LIN {X 0,Y 298.848,Z 1149.054,A -85,B 0,C 180,E1 12296.263,E2 12296.263} C_VEL
LIN {X 0,Y 306.631,Z 1138.503,A -85,B 0,C 180,E1 12292.663,E2 12292.663} C_VEL
LIN {X 0,Y 315.41,Z 1126.647,A -85,B 0,C 180,E1 12289.23,E2 12289.23} C_VEL
LIN {X 0,Y 327.193,Z 1110.564,A -85,B 0,C 180,E1 12285.344,E2 12285.344} C_VEL
LIN {X 0,Y 338.522,Z 1094.359,A -85,B 0,C 180,E1 12282.153,E2 12282.153} C_VEL
LIN {X 0,Y 348.344,Z 1079.778,A -85,B 0,C 180,E1 12279.714,E2 12279.714} C_VEL
LIN {X 0,Y 358.568,Z 1063.892,A -85,B 0,C 180,E1 12277.439,E2 12277.439} C_VEL
LIN {X 0,Y 370.942,Z 1043.552,A -85,B 0,C 180,E1 12274.974,E2 12274.974} C_VEL
LIN {X 0,Y 382.686,Z 1022.269,A -85,B 0,C 180,E1 12272.861,E2 12272.861} C_VEL
LIN {X 0,Y 392.079,Z 1003.934,A -85,B 0,C 180,E1 12271.318,E2 12271.318} C_VEL
LIN {X 0,Y 400.638,Z 985.807,A -85,B 0,C 180,E1 12270.004,E2 12270.004} C_VEL
LIN {X 0,Y 409.368,Z 965.527,A -85,B 0,C 180,E1 12268.737,E2 12268.737} C_VEL
LIN {X 0,Y 419.427,Z 939.151,A -85,B 0,C 180,E1 12267.379,E2 12267.379} C_VEL
LIN {X 0,Y 426.63,Z 917.308,A -85,B 0,C 180,E1 12266.458,E2 12266.458} C_VEL
LIN {X 0,Y 432.569,Z 896.655,A -85,B 0,C 180,E1 12265.726,E2 12265.726} C_VEL
LIN {X 0,Y 432.97,Z 895.159,A -85,B 0,C 180,E1 12265.678,E2 12265.678} C_VEL
LIN {X 0,Y 434.572,Z 887.998,A -85,B 0,C 180,E1 12265.339,E2 12265.339} C_VEL
LIN {X 0,Y 436.586,Z 870.292,A -85,B 0,C 180,E1 12264.11,E2 12264.11} C_VEL
LIN {X 0,Y 437.717,Z 862.972,A -85,B 0,C 180,E1 12263.81,E2 12263.81} C_VEL
LIN {X 0,Y 441.966,Z 839.481,A -85,B 0,C 180,E1 12263.335,E2 12263.335} C_VEL
LIN {X 0,Y 444.937,Z 817.163,A -85,B 0,C 180,E1 12262.954,E2 12262.954} C_VEL
LIN {X 0,Y 464.403,Z 606.648,A -85,B 0,C 180,E1 12259.789,E2 12259.789} C_VEL
LIN {X 0,Y 465.771,Z 591.946,A -85,B 0,C 180,E1 12259.566,E2 12259.566} C_VEL
LIN {X 0,Y 461.251,Z 583.723,A -85,B 0,C 180,E1 12256.887,E2 12256.887} C_VEL
LIN {X 0,Y 458.078,Z 578.07,A -85,B 0,C 180,E1 12254.603,E2 12254.603} C_VEL
LIN {X 0,Y 456.376,Z 575.276,A -85,B 0,C 180,E1 12253.171,E2 12253.171} C_VEL
LIN {X 0,Y 454.555,Z 571.903,A -85,B 0,C 180,E1 12251.29,E2 12251.29} C_VEL
LIN {X 0,Y 452.297,Z 567.52,A -85,B 0,C 180,E1 12247.878,E2 12247.878} C_VEL
LIN {X 0,Y 451.171,Z 566.506,A -85,B 0,C 180,E1 12243.176,E2 12243.176} C_VEL
LIN {X 0,Y 452.449,Z 567.778,A -85,B 0,C 180,E1 12238.924,E2 12238.924} C_VEL
LIN {X 0,Y 454.653,Z 571.991,A -85,B 0,C 180,E1 12235.712,E2 12235.712} C_VEL
LIN {X 0,Y 457.727,Z 577.434,A -85,B 0,C 180,E1 12232.784,E2 12232.784} C_VEL
LIN {X 0,Y 461.178,Z 583.607,A -85,B 0,C 180,E1 12230.264,E2 12230.264} C_VEL
LIN {X 0,Y 465.657,Z 591.717,A -85,B 0,C 180,E1 12227.6,E2 12227.6} C_VEL
LIN {X 0,Y 465.809,Z 592.384,A -85,B 0,C 180,E1 12227.497,E2 12227.497} C_VEL
LIN {X 0,Y 445.561,Z 812.948,A -85,B 0,C 180,E1 12224.189,E2 12224.189} C_VEL
LIN {X 0,Y 442.274,Z 839.432,A -85,B 0,C 180,E1 12223.745,E2 12223.745} C_VEL
LIN {X 0,Y 438.393,Z 861.631,A -85,B 0,C 180,E1 12223.316,E2 12223.316} C_VEL
LIN {X 0,Y 433.612,Z 883.484,A -85,B 0,C 180,E1 12222.797,E2 12222.797} C_VEL
LIN {X 0,Y 426.781,Z 909.478,A -85,B 0,C 180,E1 12222.021,E2 12222.021} C_VEL
LIN {X 0,Y 418.611,Z 934.825,A -85,B 0,C 180,E1 12221.058,E2 12221.058} C_VEL
LIN {X 0,Y 411.381,Z 954.622,A -85,B 0,C 180,E1 12220.152,E2 12220.152} C_VEL
LIN {X 0,Y 403.296,Z 974.499,A -85,B 0,C 180,E1 12219.083,E2 12219.083} C_VEL
LIN {X 0,Y 394.183,Z 994.824,A -85,B 0,C 180,E1 12217.793,E2 12217.793} C_VEL
LIN {X 0,Y 382.115,Z 1019.005,A -85,B 0,C 180,E1 12215.952,E2 12215.952} C_VEL
LIN {X 0,Y 371.516,Z 1038.231,A -85,B 0,C 180,E1 12214.189,E2 12214.189} C_VEL
LIN {X 0,Y 361.689,Z 1054.851,A -85,B 0,C 180,E1 12212.41,E2 12212.41} C_VEL
LIN {X 0,Y 351.422,Z 1071.214,A -85,B 0,C 180,E1 12210.366,E2 12210.366} C_VEL
LIN {X 0,Y 339.159,Z 1089.74,A -85,B 0,C 180,E1 12207.631,E2 12207.631} C_VEL
LIN {X 0,Y 326.616,Z 1107.457,A -85,B 0,C 180,E1 12204.432,E2 12204.432} C_VEL
LIN {X 0,Y 316.723,Z 1120.957,A -85,B 0,C 180,E1 12201.527,E2 12201.527} C_VEL
LIN {X 0,Y 307.464,Z 1133.293,A -85,B 0,C 180,E1 12198.413,E2 12198.413} C_VEL
LIN {X 0,Y 298.632,Z 1144.957,A -85,B 0,C 180,E1 12194.947,E2 12194.947} C_VEL
LIN {X 0,Y 288.909,Z 1157.956,A -85,B 0,C 180,E1 12190.328,E2 12190.328} C_VEL
LIN {X 0,Y 280.637,Z 1169.184,A -85,B 0,C 180,E1 12185.322,E2 12185.322} C_VEL
LIN {X 0,Y 275.188,Z 1177.115,A -85,B 0,C 180,E1 12181.06,E2 12181.06} C_VEL
LIN {X 0,Y 270.808,Z 1184.121,A -85,B 0,C 180,E1 12176.535,E2 12176.535} C_VEL
LIN {X 0,Y 267.412,Z 1190.479,A -85,B 0,C 180,E1 12171.495,E2 12171.495} C_VEL
LIN {X 0,Y 265.075,Z 1196.182,A -85,B 0,C 180,E1 12165.534,E2 12165.534} C_VEL
LIN {X 0,Y 264.182,Z 1199.596,A -85,B 0,C 180,E1 12160.467,E2 12160.467} C_VEL
LIN {X 0,Y 263.953,Z 1201.5,A -85,B 0,C 180,E1 12156.307,E2 12156.307} C_VEL
LIN {X 0,Y 263.915,Z 1202.584,A -85,B 0,C 180,E1 12151.954,E2 12151.954} C_VEL
LIN {X 0,Y 263.913,Z 1202.769,A -85,B 0,C 180,E1 12147.829,E2 12147.829} C_VEL
LIN {X 0,Y 263.958,Z 1202.061,A -85,B 0,C 180,E1 12143.475,E2 12143.475} C_VEL
LIN {X 0,Y 264.264,Z 1200.332,A -85,B 0,C 180,E1 12138.874,E2 12138.874} C_VEL
LIN {X 0,Y 265.245,Z 1197.443,A -85,B 0,C 180,E1 12134.027,E2 12134.027} C_VEL
LIN {X 0,Y 267.07,Z 1193.652,A -85,B 0,C 180,E1 12129.388,E2 12129.388} C_VEL
LIN {X 0,Y 269.995,Z 1188.844,A -85,B 0,C 180,E1 12124.794,E2 12124.794} C_VEL
LIN {X 0,Y 274.352,Z 1182.67,A -85,B 0,C 180,E1 12120.047,E2 12120.047} C_VEL
LIN {X 0,Y 281.35,Z 1173.897,A -85,B 0,C 180,E1 12114.601,E2 12114.601} C_VEL
LIN {X 0,Y 290.342,Z 1163.146,A -85,B 0,C 180,E1 12109.393,E2 12109.393} C_VEL
LIN {X 0,Y 299.108,Z 1153.094,A -85,B 0,C 180,E1 12105.401,E2 12105.401} C_VEL
LIN {X 0,Y 308.541,Z 1142.322,A -85,B 0,C 180,E1 12101.812,E2 12101.812} C_VEL
LIN {X 0,Y 320.174,Z 1128.958,A -85,B 0,C 180,E1 12098.098,E2 12098.098} C_VEL
LIN {X 0,Y 334.188,Z 1112.217,A -85,B 0,C 180,E1 12094.334,E2 12094.334} C_VEL
LIN {X 0,Y 346.206,Z 1097.244,A -85,B 0,C 180,E1 12091.573,E2 12091.573} C_VEL
LIN {X 0,Y 357.593,Z 1082.406,A -85,B 0,C 180,E1 12089.264,E2 12089.264} C_VEL
LIN {X 0,Y 369.525,Z 1065.998,A -85,B 0,C 180,E1 12087.101,E2 12087.101} C_VEL
LIN {X 0,Y 384.556,Z 1043.665,A -85,B 0,C 180,E1 12084.673,E2 12084.673} C_VEL
LIN {X 0,Y 395.974,Z 1025.155,A -85,B 0,C 180,E1 12083.018,E2 12083.018} C_VEL
LIN {X 0,Y 405.897,Z 1007.76,A -85,B 0,C 180,E1 12081.686,E2 12081.686} C_VEL
LIN {X 0,Y 415.681,Z 989.14,A -85,B 0,C 180,E1 12080.466,E2 12080.466} C_VEL
LIN {X 0,Y 425.434,Z 968.768,A -85,B 0,C 180,E1 12079.334,E2 12079.334} C_VEL
LIN {X 0,Y 436.603,Z 942.294,A -85,B 0,C 180,E1 12078.125,E2 12078.125} C_VEL
LIN {X 0,Y 444.581,Z 920.371,A -85,B 0,C 180,E1 12077.313,E2 12077.313} C_VEL
LIN {X 0,Y 451.161,Z 899.649,A -85,B 0,C 180,E1 12076.676,E2 12076.676} C_VEL
LIN {X 0,Y 456.952,Z 878.361,A -85,B 0,C 180,E1 12076.135,E2 12076.135} C_VEL
LIN {X 0,Y 462.441,Z 854.005,A -85,B 0,C 180,E1 12075.644,E2 12075.644} C_VEL
LIN {X 0,Y 467.168,Z 825.022,A -85,B 0,C 180,E1 12075.163,E2 12075.163} C_VEL
LIN {X 0,Y 474.721,Z 753.481,A -85,B 0,C 180,E1 12074.115,E2 12074.115} C_VEL
LIN {X 0,Y 489.723,Z 608.892,A -85,B 0,C 180,E1 12072.02,E2 12072.02} C_VEL
LIN {X 0,Y 487.951,Z 605.447,A -85,B 0,C 180,E1 12070.15,E2 12070.15} C_VEL
LIN {X 0,Y 486.244,Z 601.834,A -85,B 0,C 180,E1 12067.562,E2 12067.562} C_VEL
LIN {X 0,Y 485.116,Z 600.297,A -85,B 0,C 180,E1 12063.427,E2 12063.427} C_VEL
LIN {X 0,Y 485.932,Z 601.575,A -85,B 0,C 180,E1 12059.822,E2 12059.822} C_VEL
LIN {X 0,Y 486.458,Z 602.272,A -85,B 0,C 180,E1 12058.822,E2 12058.822} C_VEL
LIN {X 0,Y 488.722,Z 606.921,A -85,B 0,C 180,E1 12055.776,E2 12055.776} C_VEL
LIN {X 0,Y 489.67,Z 609.104,A -85,B 0,C 180,E1 12054.794,E2 12054.794} C_VEL
LIN {X 0,Y 467.761,Z 819.218,A -85,B 0,C 180,E1 12051.761,E2 12051.761} C_VEL
LIN {X 0,Y 464.351,Z 842.109,A -85,B 0,C 180,E1 12051.392,E2 12051.392} C_VEL
LIN {X 0,Y 458.756,Z 869.685,A -85,B 0,C 180,E1 12050.863,E2 12050.863} C_VEL
LIN {X 0,Y 452.233,Z 894.407,A -85,B 0,C 180,E1 12050.238,E2 12050.238} C_VEL
LIN {X 0,Y 445.762,Z 915.186,A -85,B 0,C 180,E1 12049.598,E2 12049.598} C_VEL
LIN {X 0,Y 438.233,Z 936.245,A -85,B 0,C 180,E1 12048.817,E2 12048.817} C_VEL
LIN {X 0,Y 428.413,Z 960.404,A -85,B 0,C 180,E1 12047.738,E2 12047.738} C_VEL
LIN {X 0,Y 417.012,Z 984.563,A -85,B 0,C 180,E1 12046.409,E2 12046.409} C_VEL
LIN {X 0,Y 407.061,Z 1003.571,A -85,B 0,C 180,E1 12045.165,E2 12045.165} C_VEL
LIN {X 0,Y 396.757,Z 1021.657,A -85,B 0,C 180,E1 12043.77,E2 12043.77} C_VEL
LIN {X 0,Y 385.992,Z 1039.101,A -85,B 0,C 180,E1 12042.201,E2 12042.201} C_VEL
LIN {X 0,Y 371.615,Z 1060.6,A -85,B 0,C 180,E1 12039.886,E2 12039.886} C_VEL
LIN {X 0,Y 358.628,Z 1078.377,A -85,B 0,C 180,E1 12037.544,E2 12037.544} C_VEL
LIN {X 0,Y 347.334,Z 1092.999,A -85,B 0,C 180,E1 12035.26,E2 12035.26} C_VEL
LIN {X 0,Y 336.246,Z 1106.691,A -85,B 0,C 180,E1 12032.745,E2 12032.745} C_VEL
LIN {X 0,Y 323.776,Z 1121.525,A -85,B 0,C 180,E1 12029.495,E2 12029.495} C_VEL
LIN {X 0,Y 310.177,Z 1137.009,A -85,B 0,C 180,E1 12025.285,E2 12025.285} C_VEL
LIN {X 0,Y 300.104,Z 1148.266,A -85,B 0,C 180,E1 12021.531,E2 12021.531} C_VEL
LIN {X 0,Y 291.682,Z 1157.706,A -85,B 0,C 180,E1 12017.768,E2 12017.768} C_VEL
LIN {X 0,Y 283.4,Z 1167.233,A -85,B 0,C 180,E1 12013.192,E2 12013.192} C_VEL
LIN {X 0,Y 275.392,Z 1176.9,A -85,B 0,C 180,E1 12007.324,E2 12007.324} C_VEL
LIN {X 0,Y 270.615,Z 1183.268,A -85,B 0,C 180,E1 12002.394,E2 12002.394} C_VEL
LIN {X 0,Y 267.55,Z 1187.968,A -85,B 0,C 180,E1 11997.849,E2 11997.849} C_VEL
LIN {X 0,Y 265.565,Z 1191.67,A -85,B 0,C 180,E1 11993.263,E2 11993.263} C_VEL
LIN {X 0,Y 264.48,Z 1194.36,A -85,B 0,C 180,E1 11988.744,E2 11988.744} C_VEL
LIN {X 0,Y 264.052,Z 1196.046,A -85,B 0,C 180,E1 11984.472,E2 11984.472} C_VEL
LIN {X 0,Y 263.934,Z 1196.873,A -85,B 0,C 180,E1 11980.477,E2 11980.477} C_VEL
LIN {X 0,Y 263.92,Z 1196.969,A -85,B 0,C 180,E1 11976.526,E2 11976.526} C_VEL
LIN {X 0,Y 263.936,Z 1196.281,A -85,B 0,C 180,E1 11972.388,E2 11972.388} C_VEL
LIN {X 0,Y 264.123,Z 1194.682,A -85,B 0,C 180,E1 11968.048,E2 11968.048} C_VEL
LIN {X 0,Y 264.764,Z 1191.92,A -85,B 0,C 180,E1 11963.332,E2 11963.332} C_VEL
LIN {X 0,Y 266.139,Z 1188.198,A -85,B 0,C 180,E1 11958.734,E2 11958.734} C_VEL
LIN {X 0,Y 268.44,Z 1183.501,A -85,B 0,C 180,E1 11954.223,E2 11954.223} C_VEL
LIN {X 0,Y 271.793,Z 1177.722,A -85,B 0,C 180,E1 11949.738,E2 11949.738} C_VEL
LIN {X 0,Y 276.754,Z 1170.251,A -85,B 0,C 180,E1 11944.995,E2 11944.995} C_VEL
LIN {X 0,Y 284.886,Z 1159.006,A -85,B 0,C 180,E1 11939.306,E2 11939.306} C_VEL
LIN {X 0,Y 292.503,Z 1148.942,A -85,B 0,C 180,E1 11935.19,E2 11935.19} C_VEL
LIN {X 0,Y 300.637,Z 1138.364,A -85,B 0,C 180,E1 11931.543,E2 11931.543} C_VEL
LIN {X 0,Y 310.272,Z 1125.864,A -85,B 0,C 180,E1 11927.911,E2 11927.911} C_VEL
LIN {X 0,Y 323.096,Z 1108.838,A -85,B 0,C 180,E1 11923.859,E2 11923.859} C_VEL
LIN {X 0,Y 333.735,Z 1094.099,A -85,B 0,C 180,E1 11920.976,E2 11920.976} C_VEL
LIN {X 0,Y 343.862,Z 1079.484,A -85,B 0,C 180,E1 11918.54,E2 11918.54} C_VEL
LIN {X 0,Y 354.807,Z 1062.9,A -85,B 0,C 180,E1 11916.185,E2 11916.185} C_VEL
LIN {X 0,Y 367.89,Z 1041.698,A -85,B 0,C 180,E1 11913.673,E2 11913.673} C_VEL
LIN {X 0,Y 379.107,Z 1021.786,A -85,B 0,C 180,E1 11911.727,E2 11911.727} C_VEL
LIN {X 0,Y 388.71,Z 1003.39,A -85,B 0,C 180,E1 11910.201,E2 11910.201} C_VEL
LIN {X 0,Y 397.461,Z 985.186,A -85,B 0,C 180,E1 11908.904,E2 11908.904} C_VEL
LIN {X 0,Y 407.502,Z 962.18,A -85,B 0,C 180,E1 11907.503,E2 11907.503} C_VEL
LIN {X 0,Y 417,Z 937.133,A -85,B 0,C 180,E1 11906.266,E2 11906.266} C_VEL
LIN {X 0,Y 423.95,Z 916.256,A -85,B 0,C 180,E1 11905.408,E2 11905.408} C_VEL
LIN {X 0,Y 430,Z 895.421,A -85,B 0,C 180,E1 11904.689,E2 11904.689} C_VEL
LIN {X 0,Y 435.648,Z 872.626,A -85,B 0,C 180,E1 11904.044,E2 11904.044} C_VEL
LIN {X 0,Y 437.717,Z 862.972,A -85,B 0,C 180,E1 11903.81,E2 11903.81} C_VEL
LIN {X 0,Y 438.835,Z 855.588,A -85,B 0,C 180,E1 11903.525,E2 11903.525} C_VEL
LIN {X 0,Y 440.138,Z 836.289,A -85,B 0,C 180,E1 11902.384,E2 11902.384} C_VEL
LIN {X 0,Y 440.881,Z 829.878,A -85,B 0,C 180,E1 11902.177,E2 11902.177} C_VEL
LIN {X 0,Y 444.973,Z 790.912,A -85,B 0,C 180,E1 11901.569,E2 11901.569} C_VEL
LIN {X 0,Y 463.11,Z 597.491,A -85,B 0,C 180,E1 11898.684,E2 11898.684} C_VEL
LIN {X 0,Y 459.071,Z 590.031,A -85,B 0,C 180,E1 11896.123,E2 11896.123} C_VEL
LIN {X 0,Y 456.096,Z 584.401,A -85,B 0,C 180,E1 11893.797,E2 11893.797} C_VEL
LIN {X 0,Y 453.353,Z 579.65,A -85,B 0,C 180,E1 11891.058,E2 11891.058} C_VEL
LIN {X 0,Y 451.257,Z 575.43,A -85,B 0,C 180,E1 11887.768,E2 11887.768} C_VEL
LIN {X 0,Y 450.201,Z 574.441,A -85,B 0,C 180,E1 11883.056,E2 11883.056} C_VEL
LIN {X 0,Y 451.425,Z 575.768,A -85,B 0,C 180,E1 11878.985,E2 11878.985} C_VEL
LIN {X 0,Y 453.984,Z 580.782,A -85,B 0,C 180,E1 11875.326,E2 11875.326} C_VEL
LIN {X 0,Y 456.496,Z 585.256,A -85,B 0,C 180,E1 11872.954,E2 11872.954} C_VEL
LIN {X 0,Y 460.172,Z 591.885,A -85,B 0,C 180,E1 11870.242,E2 11870.242} C_VEL
LIN {X 0,Y 463.183,Z 597.705,A -85,B 0,C 180,E1 11868.373,E2 11868.373} C_VEL
LIN {X 0,Y 442.631,Z 816.279,A -85,B 0,C 180,E1 11865.117,E2 11865.117} C_VEL
LIN {X 0,Y 439.544,Z 840.175,A -85,B 0,C 180,E1 11864.717,E2 11864.717} C_VEL
LIN {X 0,Y 435.587,Z 862.291,A -85,B 0,C 180,E1 11864.295,E2 11864.295} C_VEL
LIN {X 0,Y 430.468,Z 885.146,A -85,B 0,C 180,E1 11863.756,E2 11863.756} C_VEL
LIN {X 0,Y 422.635,Z 913.497,A -85,B 0,C 180,E1 11862.895,E2 11862.895} C_VEL
LIN {X 0,Y 415.288,Z 935.737,A -85,B 0,C 180,E1 11862.05,E2 11862.05} C_VEL
LIN {X 0,Y 407.832,Z 955.7,A -85,B 0,C 180,E1 11861.143,E2 11861.143} C_VEL
LIN {X 0,Y 399.392,Z 975.958,A -85,B 0,C 180,E1 11860.059,E2 11860.059} C_VEL
LIN {X 0,Y 388.385,Z 999.758,A -85,B 0,C 180,E1 11858.535,E2 11858.535} C_VEL
LIN {X 0,Y 376.89,Z 1021.741,A -85,B 0,C 180,E1 11856.814,E2 11856.814} C_VEL
LIN {X 0,Y 367.17,Z 1038.915,A -85,B 0,C 180,E1 11855.235,E2 11855.235} C_VEL
LIN {X 0,Y 357.183,Z 1055.378,A -85,B 0,C 180,E1 11853.475,E2 11853.475} C_VEL
LIN {X 0,Y 346.007,Z 1072.703,A -85,B 0,C 180,E1 11851.302,E2 11851.302} C_VEL
LIN {X 0,Y 331.792,Z 1093.31,A -85,B 0,C 180,E1 11848.171,E2 11848.171} C_VEL
LIN {X 0,Y 320.741,Z 1108.389,A -85,B 0,C 180,E1 11845.384,E2 11845.384} C_VEL
LIN {X 0,Y 310.954,Z 1121.299,A -85,B 0,C 180,E1 11842.573,E2 11842.573} C_VEL
LIN {X 0,Y 301.399,Z 1133.582,A -85,B 0,C 180,E1 11839.436,E2 11839.436} C_VEL
LIN {X 0,Y 291.791,Z 1145.799,A -85,B 0,C 180,E1 11835.738,E2 11835.738} C_VEL
LIN {X 0,Y 280.975,Z 1159.554,A -85,B 0,C 180,E1 11830.633,E2 11830.633} C_VEL
LIN {X 0,Y 273.407,Z 1169.459,A -85,B 0,C 180,E1 11826.07,E2 11826.07} C_VEL
LIN {X 0,Y 267.786,Z 1177.242,A -85,B 0,C 180,E1 11821.767,E2 11821.767} C_VEL
LIN {X 0,Y 263.183,Z 1184.219,A -85,B 0,C 180,E1 11817.122,E2 11817.122} C_VEL
LIN {X 0,Y 259.356,Z 1191.071,A -85,B 0,C 180,E1 11811.484,E2 11811.484} C_VEL
LIN {X 0,Y 257.071,Z 1196.358,A -85,B 0,C 180,E1 11805.567,E2 11805.567} C_VEL
LIN {X 0,Y 256.213,Z 1199.464,A -85,B 0,C 180,E1 11800.796,E2 11800.796} C_VEL
LIN {X 0,Y 255.953,Z 1201.455,A -85,B 0,C 180,E1 11796.279,E2 11796.279} C_VEL
LIN {X 0,Y 255.915,Z 1202.488,A -85,B 0,C 180,E1 11792.015,E2 11792.015} C_VEL
LIN {X 0,Y 255.913,Z 1202.689,A -85,B 0,C 180,E1 11787.761,E2 11787.761} C_VEL
LIN {X 0,Y 255.97,Z 1201.929,A -85,B 0,C 180,E1 11783.045,E2 11783.045} C_VEL
LIN {X 0,Y 256.334,Z 1200.153,A -85,B 0,C 180,E1 11778.262,E2 11778.262} C_VEL
LIN {X 0,Y 257.38,Z 1197.414,A -85,B 0,C 180,E1 11773.526,E2 11773.526} C_VEL
LIN {X 0,Y 259.356,Z 1193.649,A -85,B 0,C 180,E1 11768.753,E2 11768.753} C_VEL
LIN {X 0,Y 262.509,Z 1188.849,A -85,B 0,C 180,E1 11764.017,E2 11764.017} C_VEL
LIN {X 0,Y 266.91,Z 1183.002,A -85,B 0,C 180,E1 11759.372,E2 11759.372} C_VEL
LIN {X 0,Y 272.969,Z 1175.708,A -85,B 0,C 180,E1 11754.638,E2 11754.638} C_VEL
LIN {X 0,Y 282.438,Z 1165.063,A -85,B 0,C 180,E1 11749.087,E2 11749.087} C_VEL
LIN {X 0,Y 292.714,Z 1153.752,A -85,B 0,C 180,E1 11744.447,E2 11744.447} C_VEL
LIN {X 0,Y 302.503,Z 1143.04,A -85,B 0,C 180,E1 11740.808,E2 11740.808} C_VEL
LIN {X 0,Y 313.371,Z 1131.023,A -85,B 0,C 180,E1 11737.395,E2 11737.395} C_VEL
LIN {X 0,Y 327.077,Z 1115.493,A -85,B 0,C 180,E1 11733.748,E2 11733.748} C_VEL
LIN {X 0,Y 341.275,Z 1098.356,A -85,B 0,C 180,E1 11730.532,E2 11730.532} C_VEL
LIN {X 0,Y 352.932,Z 1083.631,A -85,B 0,C 180,E1 11728.229,E2 11728.229} C_VEL
LIN {X 0,Y 364.759,Z 1067.847,A -85,B 0,C 180,E1 11726.14,E2 11726.14} C_VEL
LIN {X 0,Y 377.427,Z 1049.832,A -85,B 0,C 180,E1 11724.129,E2 11724.129} C_VEL
LIN {X 0,Y 391.698,Z 1027.619,A -85,B 0,C 180,E1 11722.089,E2 11722.089} C_VEL
LIN {X 0,Y 402.823,Z 1008.606,A -85,B 0,C 180,E1 11720.639,E2 11720.639} C_VEL
LIN {X 0,Y 412.937,Z 989.771,A -85,B 0,C 180,E1 11719.42,E2 11719.42} C_VEL
LIN {X 0,Y 422.517,Z 970.179,A -85,B 0,C 180,E1 11718.346,E2 11718.346} C_VEL
LIN {X 0,Y 433.351,Z 945.415,A -85,B 0,C 180,E1 11717.214,E2 11717.214} C_VEL
LIN {X 0,Y 442.286,Z 921.417,A -85,B 0,C 180,E1 11716.332,E2 11716.332} C_VEL
LIN {X 0,Y 449.171,Z 900.148,A -85,B 0,C 180,E1 11715.689,E2 11715.689} C_VEL
LIN {X 0,Y 455.048,Z 878.936,A -85,B 0,C 180,E1 11715.16,E2 11715.16} C_VEL
LIN {X 0,Y 460.325,Z 856.02,A -85,B 0,C 180,E1 11714.705,E2 11714.705} C_VEL
LIN {X 0,Y 465.493,Z 825.554,A -85,B 0,C 180,E1 11714.204,E2 11714.204} C_VEL
LIN {X 0,Y 472.341,Z 762.313,A -85,B 0,C 180,E1 11713.286,E2 11713.286} C_VEL
LIN {X 0,Y 487.877,Z 615.419,A -85,B 0,C 180,E1 11711.197,E2 11711.197} C_VEL
LIN {X 0,Y 486.678,Z 613.023,A -85,B 0,C 180,E1 11709.818,E2 11709.818} C_VEL
LIN {X 0,Y 485.205,Z 609.734,A -85,B 0,C 180,E1 11707.46,E2 11707.46} C_VEL
LIN {X 0,Y 484.142,Z 608.225,A -85,B 0,C 180,E1 11703.315,E2 11703.315} C_VEL
LIN {X 0,Y 485.295,Z 609.813,A -85,B 0,C 180,E1 11699.174,E2 11699.174} C_VEL
LIN {X 0,Y 487.562,Z 614.715,A -85,B 0,C 180,E1 11695.943,E2 11695.943} C_VEL
LIN {X 0,Y 487.815,Z 615.548,A -85,B 0,C 180,E1 11695.636,E2 11695.636} C_VEL
LIN {X 0,Y 465.995,Z 820.655,A -85,B 0,C 180,E1 11692.706,E2 11692.706} C_VEL
LIN {X 0,Y 462.095,Z 845.781,A -85,B 0,C 180,E1 11692.304,E2 11692.304} C_VEL
LIN {X 0,Y 455.964,Z 873.94,A -85,B 0,C 180,E1 11691.751,E2 11691.751} C_VEL
LIN {X 0,Y 449.996,Z 895.916,A -85,B 0,C 180,E1 11691.197,E2 11691.197} C_VEL
LIN {X 0,Y 443.429,Z 916.521,A -85,B 0,C 180,E1 11690.57,E2 11690.57} C_VEL
LIN {X 0,Y 435.816,Z 937.363,A -85,B 0,C 180,E1 11689.807,E2 11689.807} C_VEL
LIN {X 0,Y 425.211,Z 962.757,A -85,B 0,C 180,E1 11688.68,E2 11688.68} C_VEL
LIN {X 0,Y 414.342,Z 985.231,A -85,B 0,C 180,E1 11687.456,E2 11687.456} C_VEL
LIN {X 0,Y 404.08,Z 1004.424,A -85,B 0,C 180,E1 11686.216,E2 11686.216} C_VEL
LIN {X 0,Y 393.469,Z 1022.632,A -85,B 0,C 180,E1 11684.826,E2 11684.826} C_VEL
LIN {X 0,Y 380.591,Z 1042.975,A -85,B 0,C 180,E1 11682.993,E2 11682.993} C_VEL
LIN {X 0,Y 366.412,Z 1063.233,A -85,B 0,C 180,E1 11680.762,E2 11680.762} C_VEL
LIN {X 0,Y 354.454,Z 1079.15,A -85,B 0,C 180,E1 11678.66,E2 11678.66} C_VEL
LIN {X 0,Y 342.721,Z 1093.899,A -85,B 0,C 180,E1 11676.357,E2 11676.357} C_VEL
LIN {X 0,Y 330.129,Z 1108.948,A -85,B 0,C 180,E1 11673.562,E2 11673.562} C_VEL
LIN {X 0,Y 315.133,Z 1125.965,A -85,B 0,C 180,E1 11669.655,E2 11669.655} C_VEL
LIN {X 0,Y 304.036,Z 1138.054,A -85,B 0,C 180,E1 11666.234,E2 11666.234} C_VEL
LIN {X 0,Y 294.231,Z 1148.574,A -85,B 0,C 180,E1 11662.672,E2 11662.672} C_VEL
LIN {X 0,Y 284.993,Z 1158.455,A -85,B 0,C 180,E1 11658.659,E2 11658.659} C_VEL
LIN {X 0,Y 275.319,Z 1169.106,A -85,B 0,C 180,E1 11653.344,E2 11653.344} C_VEL
LIN {X 0,Y 267.721,Z 1177.73,A -85,B 0,C 180,E1 11647.77,E2 11647.77} C_VEL
LIN {X 0,Y 262.966,Z 1183.719,A -85,B 0,C 180,E1 11642.937,E2 11642.937} C_VEL
LIN {X 0,Y 259.61,Z 1188.559,A -85,B 0,C 180,E1 11638.026,E2 11638.026} C_VEL
LIN {X 0,Y 257.357,Z 1192.611,A -85,B 0,C 180,E1 11632.62,E2 11632.62} C_VEL
LIN {X 0,Y 256.215,Z 1195.623,A -85,B 0,C 180,E1 11626.551,E2 11626.551} C_VEL
LIN {X 0,Y 255.946,Z 1196.882,A -85,B 0,C 180,E1 11621.492,E2 11621.492} C_VEL
LIN {X 0,Y 255.925,Z 1197.094,A -85,B 0,C 180,E1 11616.956,E2 11616.956} C_VEL
LIN {X 0,Y 255.936,Z 1196.409,A -85,B 0,C 180,E1 11612.463,E2 11612.463} C_VEL
LIN {X 0,Y 256.147,Z 1194.724,A -85,B 0,C 180,E1 11607.763,E2 11607.763} C_VEL
LIN {X 0,Y 256.815,Z 1192.063,A -85,B 0,C 180,E1 11603.068,E2 11603.068} C_VEL
LIN {X 0,Y 258.255,Z 1188.409,A -85,B 0,C 180,E1 11598.386,E2 11598.386} C_VEL
LIN {X 0,Y 260.689,Z 1183.74,A -85,B 0,C 180,E1 11593.741,E2 11593.741} C_VEL
LIN {X 0,Y 264.193,Z 1178.029,A -85,B 0,C 180,E1 11589.161,E2 11589.161} C_VEL
LIN {X 0,Y 269.169,Z 1170.891,A -85,B 0,C 180,E1 11584.476,E2 11584.476} C_VEL
LIN {X 0,Y 277.115,Z 1160.456,A -85,B 0,C 180,E1 11578.939,E2 11578.939} C_VEL
LIN {X 0,Y 285.952,Z 1149.215,A -85,B 0,C 180,E1 11574.217,E2 11574.217} C_VEL
LIN {X 0,Y 294.316,Z 1138.783,A -85,B 0,C 180,E1 11570.559,E2 11570.559} C_VEL
LIN {X 0,Y 303.298,Z 1127.554,A -85,B 0,C 180,E1 11567.227,E2 11567.227} C_VEL
LIN {X 0,Y 314.946,Z 1112.769,A -85,B 0,C 180,E1 11563.546,E2 11563.546} C_VEL
LIN {X 0,Y 328.02,Z 1095.319,A -85,B 0,C 180,E1 11560.03,E2 11560.03} C_VEL
LIN {X 0,Y 338.898,Z 1080.087,A -85,B 0,C 180,E1 11557.474,E2 11557.474} C_VEL
LIN {X 0,Y 349.516,Z 1064.448,A -85,B 0,C 180,E1 11555.242,E2 11555.242} C_VEL
LIN {X 0,Y 361.981,Z 1044.961,A -85,B 0,C 180,E1 11552.892,E2 11552.892} C_VEL
LIN {X 0,Y 374.609,Z 1023.252,A -85,B 0,C 180,E1 11550.746,E2 11550.746} C_VEL
LIN {X 0,Y 384.761,Z 1004.269,A -85,B 0,C 180,E1 11549.174,E2 11549.174} C_VEL
LIN {X 0,Y 393.679,Z 986.144,A -85,B 0,C 180,E1 11547.891,E2 11547.891} C_VEL
LIN {X 0,Y 402.747,Z 965.871,A -85,B 0,C 180,E1 11546.654,E2 11546.654} C_VEL
LIN {X 0,Y 413.177,Z 939.527,A -85,B 0,C 180,E1 11545.333,E2 11545.333} C_VEL
LIN {X 0,Y 420.722,Z 917.399,A -85,B 0,C 180,E1 11544.427,E2 11544.427} C_VEL
LIN {X 0,Y 426.971,Z 896.339,A -85,B 0,C 180,E1 11543.706,E2 11543.706} C_VEL
LIN {X 0,Y 432.496,Z 874.558,A -85,B 0,C 180,E1 11543.093,E2 11543.093} C_VEL
LIN {X 0,Y 438.082,Z 847.644,A -85,B 0,C 180,E1 11542.494,E2 11542.494} C_VEL
LIN {X 0,Y 440.881,Z 829.878,A -85,B 0,C 180,E1 11542.177,E2 11542.177} C_VEL
LIN {X 0,Y 441.632,Z 822.395,A -85,B 0,C 180,E1 11541.928,E2 11541.928} C_VEL
LIN {X 0,Y 441.723,Z 802.826,A -85,B 0,C 180,E1 11540.851,E2 11540.851} C_VEL
LIN {X 0,Y 442.089,Z 796.338,A -85,B 0,C 180,E1 11540.659,E2 11540.659} C_VEL
LIN {X 0,Y 460.588,Z 603.061,A -85,B 0,C 180,E1 11537.808,E2 11537.808} C_VEL
LIN {X 0,Y 456.266,Z 594.858,A -85,B 0,C 180,E1 11534.792,E2 11534.792} C_VEL
LIN {X 0,Y 454.147,Z 591.116,A -85,B 0,C 180,E1 11532.978,E2 11532.978} C_VEL
LIN {X 0,Y 452.165,Z 587.403,A -85,B 0,C 180,E1 11530.834,E2 11530.834} C_VEL
LIN {X 0,Y 450.219,Z 583.341,A -85,B 0,C 180,E1 11527.658,E2 11527.658} C_VEL
LIN {X 0,Y 449.223,Z 582.381,A -85,B 0,C 180,E1 11523.062,E2 11523.062} C_VEL
LIN {X 0,Y 450.375,Z 583.654,A -85,B 0,C 180,E1 11519.11,E2 11519.11} C_VEL
LIN {X 0,Y 452.817,Z 588.579,A -85,B 0,C 180,E1 11515.504,E2 11515.504} C_VEL
LIN {X 0,Y 455.269,Z 593.076,A -85,B 0,C 180,E1 11513.125,E2 11513.125} C_VEL
LIN {X 0,Y 458.785,Z 599.602,A -85,B 0,C 180,E1 11510.466,E2 11510.466} C_VEL
LIN {X 0,Y 460.626,Z 603.453,A -85,B 0,C 180,E1 11509.253,E2 11509.253} C_VEL
LIN {X 0,Y 439.895,Z 818.941,A -85,B 0,C 180,E1 11506.068,E2 11506.068} C_VEL
LIN {X 0,Y 436.866,Z 841.391,A -85,B 0,C 180,E1 11505.693,E2 11505.693} C_VEL
LIN {X 0,Y 432.699,Z 863.996,A -85,B 0,C 180,E1 11505.264,E2 11505.264} C_VEL
LIN {X 0,Y 426.438,Z 890.854,A -85,B 0,C 180,E1 11504.623,E2 11504.623} C_VEL
LIN {X 0,Y 419.065,Z 916.036,A -85,B 0,C 180,E1 11503.838,E2 11503.838} C_VEL
LIN {X 0,Y 412.287,Z 936.096,A -85,B 0,C 180,E1 11503.08,E2 11503.08} C_VEL
LIN {X 0,Y 404.714,Z 955.994,A -85,B 0,C 180,E1 11502.189,E2 11502.189} C_VEL
LIN {X 0,Y 395.826,Z 976.906,A -85,B 0,C 180,E1 11501.082,E2 11501.082} C_VEL
LIN {X 0,Y 383.888,Z 1001.901,A -85,B 0,C 180,E1 11499.479,E2 11499.479} C_VEL
LIN {X 0,Y 373.292,Z 1021.739,A -85,B 0,C 180,E1 11497.934,E2 11497.934} C_VEL
LIN {X 0,Y 363.397,Z 1038.84,A -85,B 0,C 180,E1 11496.379,E2 11496.379} C_VEL
LIN {X 0,Y 352.805,Z 1055.899,A -85,B 0,C 180,E1 11494.568,E2 11494.568} C_VEL
LIN {X 0,Y 340.964,Z 1073.776,A -85,B 0,C 180,E1 11492.325,E2 11492.325} C_VEL
LIN {X 0,Y 326.685,Z 1093.812,A -85,B 0,C 180,E1 11489.26,E2 11489.26} C_VEL
LIN {X 0,Y 315.396,Z 1108.751,A -85,B 0,C 180,E1 11486.486,E2 11486.486} C_VEL
LIN {X 0,Y 305.198,Z 1121.76,A -85,B 0,C 180,E1 11483.63,E2 11483.63} C_VEL
LIN {X 0,Y 294.912,Z 1134.518,A -85,B 0,C 180,E1 11480.319,E2 11480.319} C_VEL
LIN {X 0,Y 283.177,Z 1148.921,A -85,B 0,C 180,E1 11475.788,E2 11475.788} C_VEL
LIN {X 0,Y 273.312,Z 1160.836,A -85,B 0,C 180,E1 11471.093,E2 11471.093} C_VEL
LIN {X 0,Y 266.253,Z 1169.693,A -85,B 0,C 180,E1 11466.879,E2 11466.879} C_VEL
LIN {X 0,Y 260.133,Z 1177.778,A -85,B 0,C 180,E1 11462.26,E2 11462.26} C_VEL
LIN {X 0,Y 254.647,Z 1185.868,A -85,B 0,C 180,E1 11456.591,E2 11456.591} C_VEL
LIN {X 0,Y 250.81,Z 1192.492,A -85,B 0,C 180,E1 11450.469,E2 11450.469} C_VEL
LIN {X 0,Y 249.042,Z 1196.599,A -85,B 0,C 180,E1 11445.508,E2 11445.508} C_VEL
LIN {X 0,Y 248.199,Z 1199.564,A -85,B 0,C 180,E1 11440.679,E2 11440.679} C_VEL
LIN {X 0,Y 247.952,Z 1201.411,A -85,B 0,C 180,E1 11436.25,E2 11436.25} C_VEL
LIN {X 0,Y 247.916,Z 1202.415,A -85,B 0,C 180,E1 11431.849,E2 11431.849} C_VEL
LIN {X 0,Y 247.914,Z 1202.587,A -85,B 0,C 180,E1 11427.457,E2 11427.457} C_VEL
LIN {X 0,Y 247.982,Z 1201.832,A -85,B 0,C 180,E1 11422.703,E2 11422.703} C_VEL
LIN {X 0,Y 248.378,Z 1200.125,A -85,B 0,C 180,E1 11417.917,E2 11417.917} C_VEL
LIN {X 0,Y 249.532,Z 1197.387,A -85,B 0,C 180,E1 11412.992,E2 11412.992} C_VEL
LIN {X 0,Y 251.681,Z 1193.64,A -85,B 0,C 180,E1 11408.072,E2 11408.072} C_VEL
LIN {X 0,Y 255.063,Z 1188.866,A -85,B 0,C 180,E1 11403.205,E2 11403.205} C_VEL
LIN {X 0,Y 259.765,Z 1183.036,A -85,B 0,C 180,E1 11398.434,E2 11398.434} C_VEL
LIN {X 0,Y 266.457,Z 1175.478,A -85,B 0,C 180,E1 11393.422,E2 11393.422} C_VEL
LIN {X 0,Y 276.996,Z 1164.257,A -85,B 0,C 180,E1 11387.546,E2 11387.546} C_VEL
LIN {X 0,Y 286.9,Z 1153.879,A -85,B 0,C 180,E1 11383.25,E2 11383.25} C_VEL
LIN {X 0,Y 297.092,Z 1143.197,A -85,B 0,C 180,E1 11379.584,E2 11379.584} C_VEL
LIN {X 0,Y 308.323,Z 1131.252,A -85,B 0,C 180,E1 11376.173,E2 11376.173} C_VEL
LIN {X 0,Y 322.528,Z 1115.722,A -85,B 0,C 180,E1 11372.519,E2 11372.519} C_VEL
LIN {X 0,Y 337.361,Z 1098.377,A -85,B 0,C 180,E1 11369.277,E2 11369.277} C_VEL
LIN {X 0,Y 349.106,Z 1083.948,A -85,B 0,C 180,E1 11367.037,E2 11367.037} C_VEL
LIN {X 0,Y 361.216,Z 1068.207,A -85,B 0,C 180,E1 11364.97,E2 11364.97} C_VEL
LIN {X 0,Y 373.387,Z 1051.325,A -85,B 0,C 180,E1 11363.1,E2 11363.1} C_VEL
LIN {X 0,Y 388.321,Z 1028.779,A -85,B 0,C 180,E1 11361.034,E2 11361.034} C_VEL
LIN {X 0,Y 400.029,Z 1009.208,A -85,B 0,C 180,E1 11359.559,E2 11359.559} C_VEL
LIN {X 0,Y 410.333,Z 990.402,A -85,B 0,C 180,E1 11358.361,E2 11358.361} C_VEL
LIN {X 0,Y 419.979,Z 971.067,A -85,B 0,C 180,E1 11357.317,E2 11357.317} C_VEL
LIN {X 0,Y 429.762,Z 949.256,A -85,B 0,C 180,E1 11356.327,E2 11356.327} C_VEL
LIN {X 0,Y 440.121,Z 922.475,A -85,B 0,C 180,E1 11355.341,E2 11355.341} C_VEL
LIN {X 0,Y 447.315,Z 900.653,A -85,B 0,C 180,E1 11354.693,E2 11354.693} C_VEL
LIN {X 0,Y 453.277,Z 879.51,A -85,B 0,C 180,E1 11354.178,E2 11354.178} C_VEL
LIN {X 0,Y 458.479,Z 857.369,A -85,B 0,C 180,E1 11353.745,E2 11353.745} C_VEL
LIN {X 0,Y 463.544,Z 829.309,A -85,B 0,C 180,E1 11353.286,E2 11353.286} C_VEL
LIN {X 0,Y 468.817,Z 782.998,A -85,B 0,C 180,E1 11352.617,E2 11352.617} C_VEL
LIN {X 0,Y 486.123,Z 621.802,A -85,B 0,C 180,E1 11350.342,E2 11350.342} C_VEL
LIN {X 0,Y 484.168,Z 617.634,A -85,B 0,C 180,E1 11347.356,E2 11347.356} C_VEL
LIN {X 0,Y 483.164,Z 616.167,A -85,B 0,C 180,E1 11343.322,E2 11343.322} C_VEL
LIN {X 0,Y 484.304,Z 617.846,A -85,B 0,C 180,E1 11339.172,E2 11339.172} C_VEL
LIN {X 0,Y 486.085,Z 621.826,A -85,B 0,C 180,E1 11336.486,E2 11336.486} C_VEL
LIN {X 0,Y 464.517,Z 820.856,A -85,B 0,C 180,E1 11333.676,E2 11333.676} C_VEL
LIN {X 0,Y 460.484,Z 846.396,A -85,B 0,C 180,E1 11333.275,E2 11333.275} C_VEL
LIN {X 0,Y 454.326,Z 874.176,A -85,B 0,C 180,E1 11332.741,E2 11332.741} C_VEL
LIN {X 0,Y 448.56,Z 895.204,A -85,B 0,C 180,E1 11332.224,E2 11332.224} C_VEL
LIN {X 0,Y 441.911,Z 915.887,A -85,B 0,C 180,E1 11331.615,E2 11331.615} C_VEL
LIN {X 0,Y 434.412,Z 936.226,A -85,B 0,C 180,E1 11330.895,E2 11330.895} C_VEL
LIN {X 0,Y 425.022,Z 958.68,A -85,B 0,C 180,E1 11329.941,E2 11329.941} C_VEL
LIN {X 0,Y 413.018,Z 983.603,A -85,B 0,C 180,E1 11328.651,E2 11328.651} C_VEL
LIN {X 0,Y 402.168,Z 1003.655,A -85,B 0,C 180,E1 11327.393,E2 11327.393} C_VEL
LIN {X 0,Y 392.086,Z 1020.733,A -85,B 0,C 180,E1 11326.13,E2 11326.13} C_VEL
LIN {X 0,Y 380.842,Z 1038.283,A -85,B 0,C 180,E1 11324.623,E2 11324.623} C_VEL
LIN {X 0,Y 366.44,Z 1059.088,A -85,B 0,C 180,E1 11322.484,E2 11322.484} C_VEL
LIN {X 0,Y 351.876,Z 1078.1,A -85,B 0,C 180,E1 11320.063,E2 11320.063} C_VEL
LIN {X 0,Y 339.326,Z 1093.496,A -85,B 0,C 180,E1 11317.703,E2 11317.703} C_VEL
LIN {X 0,Y 326.688,Z 1108.18,A -85,B 0,C 180,E1 11315.015,E2 11315.015} C_VEL
LIN {X 0,Y 312.056,Z 1124.375,A -85,B 0,C 180,E1 11311.392,E2 11311.392} C_VEL
LIN {X 0,Y 299.365,Z 1137.679,A -85,B 0,C 180,E1 11307.672,E2 11307.672} C_VEL
LIN {X 0,Y 288.991,Z 1148.354,A -85,B 0,C 180,E1 11304.057,E2 11304.057} C_VEL
LIN {X 0,Y 279.734,Z 1157.801,A -85,B 0,C 180,E1 11300.217,E2 11300.217} C_VEL
LIN {X 0,Y 270.882,Z 1166.921,A -85,B 0,C 180,E1 11295.731,E2 11295.731} C_VEL
LIN {X 0,Y 261.465,Z 1177.021,A -85,B 0,C 180,E1 11289.405,E2 11289.405} C_VEL
LIN {X 0,Y 255.969,Z 1183.397,A -85,B 0,C 180,E1 11284.228,E2 11284.228} C_VEL
LIN {X 0,Y 252.301,Z 1188.196,A -85,B 0,C 180,E1 11279.322,E2 11279.322} C_VEL
LIN {X 0,Y 249.914,Z 1191.963,A -85,B 0,C 180,E1 11274.336,E2 11274.336} C_VEL
LIN {X 0,Y 248.605,Z 1194.63,A -85,B 0,C 180,E1 11269.5,E2 11269.5} C_VEL
LIN {X 0,Y 248.088,Z 1196.278,A -85,B 0,C 180,E1 11264.948,E2 11264.948} C_VEL
LIN {X 0,Y 247.936,Z 1197.067,A -85,B 0,C 180,E1 11260.691,E2 11260.691} C_VEL
LIN {X 0,Y 247.921,Z 1197.126,A -85,B 0,C 180,E1 11256.484,E2 11256.484} C_VEL
LIN {X 0,Y 247.942,Z 1196.401,A -85,B 0,C 180,E1 11252.08,E2 11252.08} C_VEL
LIN {X 0,Y 248.173,Z 1194.767,A -85,B 0,C 180,E1 11247.46,E2 11247.46} C_VEL
LIN {X 0,Y 248.91,Z 1192.087,A -85,B 0,C 180,E1 11242.615,E2 11242.615} C_VEL
LIN {X 0,Y 250.478,Z 1188.415,A -85,B 0,C 180,E1 11237.786,E2 11237.786} C_VEL
LIN {X 0,Y 253.176,Z 1183.608,A -85,B 0,C 180,E1 11232.893,E2 11232.893} C_VEL
LIN {X 0,Y 257.071,Z 1177.703,A -85,B 0,C 180,E1 11228.076,E2 11228.076} C_VEL
LIN {X 0,Y 263.028,Z 1169.745,A -85,B 0,C 180,E1 11222.817,E2 11222.817} C_VEL
LIN {X 0,Y 271.607,Z 1159.018,A -85,B 0,C 180,E1 11217.238,E2 11217.238} C_VEL
LIN {X 0,Y 280.13,Z 1148.71,A -85,B 0,C 180,E1 11212.9,E2 11212.9} C_VEL
LIN {X 0,Y 289.025,Z 1138.081,A -85,B 0,C 180,E1 11209.169,E2 11209.169} C_VEL
LIN {X 0,Y 300.002,Z 1124.904,A -85,B 0,C 180,E1 11205.314,E2 11205.314} C_VEL
LIN {X 0,Y 313.243,Z 1108.381,A -85,B 0,C 180,E1 11201.4,E2 11201.4} C_VEL
LIN {X 0,Y 323.986,Z 1094.396,A -85,B 0,C 180,E1 11198.668,E2 11198.668} C_VEL
LIN {X 0,Y 334.704,Z 1079.783,A -85,B 0,C 180,E1 11196.238,E2 11196.238} C_VEL
LIN {X 0,Y 345.953,Z 1063.611,A -85,B 0,C 180,E1 11193.956,E2 11193.956} C_VEL
LIN {X 0,Y 359.194,Z 1043.303,A -85,B 0,C 180,E1 11191.557,E2 11191.557} C_VEL
LIN {X 0,Y 371.682,Z 1022.104,A -85,B 0,C 180,E1 11189.513,E2 11189.513} C_VEL
LIN {X 0,Y 381.683,Z 1003.713,A -85,B 0,C 180,E1 11188.018,E2 11188.018} C_VEL
LIN {X 0,Y 391.17,Z 984.724,A -85,B 0,C 180,E1 11186.704,E2 11186.704} C_VEL
LIN {X 0,Y 401.989,Z 960.706,A -85,B 0,C 180,E1 11185.295,E2 11185.295} C_VEL
LIN {X 0,Y 411.44,Z 936.386,A -85,B 0,C 180,E1 11184.145,E2 11184.145} C_VEL
LIN {X 0,Y 418.446,Z 915.936,A -85,B 0,C 180,E1 11183.335,E2 11183.335} C_VEL
LIN {X 0,Y 424.68,Z 895.083,A -85,B 0,C 180,E1 11182.644,E2 11182.644} C_VEL
LIN {X 0,Y 430.892,Z 870.599,A -85,B 0,C 180,E1 11181.982,E2 11181.982} C_VEL
LIN {X 0,Y 436.437,Z 842.374,A -85,B 0,C 180,E1 11181.4,E2 11181.4} C_VEL
LIN {X 0,Y 439.709,Z 819.333,A -85,B 0,C 180,E1 11181.012,E2 11181.012} C_VEL
LIN {X 0,Y 442.089,Z 796.338,A -85,B 0,C 180,E1 11180.659,E2 11180.659} C_VEL
LIN {X 0,Y 442.508,Z 788.801,A -85,B 0,C 180,E1 11180.422,E2 11180.422} C_VEL
LIN {X 0,Y 442.645,Z 769.219,A -85,B 0,C 180,E1 11179.355,E2 11179.355} C_VEL
LIN {X 0,Y 443.071,Z 762.736,A -85,B 0,C 180,E1 11179.166,E2 11179.166} C_VEL
LIN {X 0,Y 458.13,Z 608.831,A -85,B 0,C 180,E1 11176.915,E2 11176.915} C_VEL
LIN {X 0,Y 454.431,Z 601.61,A -85,B 0,C 180,E1 11174.137,E2 11174.137} C_VEL
LIN {X 0,Y 452.706,Z 598.502,A -85,B 0,C 180,E1 11172.566,E2 11172.566} C_VEL
LIN {X 0,Y 450.982,Z 595.151,A -85,B 0,C 180,E1 11170.604,E2 11170.604} C_VEL
LIN {X 0,Y 449.182,Z 591.251,A -85,B 0,C 180,E1 11167.547,E2 11167.547} C_VEL
LIN {X 0,Y 448.246,Z 590.321,A -85,B 0,C 180,E1 11163.069,E2 11163.069} C_VEL
LIN {X 0,Y 449.327,Z 591.539,A -85,B 0,C 180,E1 11159.235,E2 11159.235} C_VEL
LIN {X 0,Y 451.655,Z 596.375,A -85,B 0,C 180,E1 11155.683,E2 11155.683} C_VEL
LIN {X 0,Y 453.995,Z 600.789,A -85,B 0,C 180,E1 11153.343,E2 11153.343} C_VEL
LIN {X 0,Y 457.405,Z 607.316,A -85,B 0,C 180,E1 11150.691,E2 11150.691} C_VEL
LIN {X 0,Y 458.172,Z 609.169,A -85,B 0,C 180,E1 11150.144,E2 11150.144} C_VEL
LIN {X 0,Y 437.46,Z 820.026,A -85,B 0,C 180,E1 11147.055,E2 11147.055} C_VEL
LIN {X 0,Y 434.359,Z 842.299,A -85,B 0,C 180,E1 11146.686,E2 11146.686} C_VEL
LIN {X 0,Y 429.842,Z 866.133,A -85,B 0,C 180,E1 11146.237,E2 11146.237} C_VEL
LIN {X 0,Y 422.827,Z 894.666,A -85,B 0,C 180,E1 11145.544,E2 11145.544} C_VEL
LIN {X 0,Y 416.128,Z 916.987,A -85,B 0,C 180,E1 11144.85,E2 11144.85} C_VEL
LIN {X 0,Y 409.112,Z 937.298,A -85,B 0,C 180,E1 11144.091,E2 11144.091} C_VEL
LIN {X 0,Y 401.108,Z 957.824,A -85,B 0,C 180,E1 11143.178,E2 11143.178} C_VEL
LIN {X 0,Y 390.337,Z 982.394,A -85,B 0,C 180,E1 11141.864,E2 11141.864} C_VEL
LIN {X 0,Y 378.964,Z 1005.032,A -85,B 0,C 180,E1 11140.374,E2 11140.374} C_VEL
LIN {X 0,Y 368.947,Z 1023.29,A -85,B 0,C 180,E1 11138.944,E2 11138.944} C_VEL
LIN {X 0,Y 358.592,Z 1040.699,A -85,B 0,C 180,E1 11137.357,E2 11137.357} C_VEL
LIN {X 0,Y 346.574,Z 1059.48,A -85,B 0,C 180,E1 11135.335,E2 11135.335} C_VEL
LIN {X 0,Y 331.889,Z 1080.584,A -85,B 0,C 180,E1 11132.552,E2 11132.552} C_VEL
LIN {X 0,Y 320.055,Z 1096.454,A -85,B 0,C 180,E1 11130.009,E2 11130.009} C_VEL
LIN {X 0,Y 308.918,Z 1110.69,A -85,B 0,C 180,E1 11127.301,E2 11127.301} C_VEL
LIN {X 0,Y 296.313,Z 1126.236,A -85,B 0,C 180,E1 11123.752,E2 11123.752} C_VEL
LIN {X 0,Y 283.776,Z 1141.009,A -85,B 0,C 180,E1 11119.557,E2 11119.557} C_VEL
LIN {X 0,Y 274.055,Z 1152.303,A -85,B 0,C 180,E1 11115.65,E2 11115.65} C_VEL
LIN {X 0,Y 265.532,Z 1162.277,A -85,B 0,C 180,E1 11111.508,E2 11111.508} C_VEL
LIN {X 0,Y 257.957,Z 1171.429,A -85,B 0,C 180,E1 11106.926,E2 11106.926} C_VEL
LIN {X 0,Y 250.043,Z 1181.617,A -85,B 0,C 180,E1 11100.52,E2 11100.52} C_VEL
LIN {X 0,Y 245.409,Z 1188.344,A -85,B 0,C 180,E1 11095.07,E2 11095.07} C_VEL
LIN {X 0,Y 242.667,Z 1193.107,A -85,B 0,C 180,E1 11090.249,E2 11090.249} C_VEL
LIN {X 0,Y 240.999,Z 1196.871,A -85,B 0,C 180,E1 11085.398,E2 11085.398} C_VEL
LIN {X 0,Y 240.205,Z 1199.561,A -85,B 0,C 180,E1 11080.768,E2 11080.768} C_VEL
LIN {X 0,Y 239.958,Z 1201.297,A -85,B 0,C 180,E1 11076.46,E2 11076.46} C_VEL
LIN {X 0,Y 239.916,Z 1202.319,A -85,B 0,C 180,E1 11071.911,E2 11071.911} C_VEL
LIN {X 0,Y 239.915,Z 1202.508,A -85,B 0,C 180,E1 11067.372,E2 11067.372} C_VEL
LIN {X 0,Y 239.988,Z 1201.803,A -85,B 0,C 180,E1 11062.575,E2 11062.575} C_VEL
LIN {X 0,Y 240.432,Z 1200.08,A -85,B 0,C 180,E1 11057.511,E2 11057.511} C_VEL
LIN {X 0,Y 241.703,Z 1197.36,A -85,B 0,C 180,E1 11052.423,E2 11052.423} C_VEL
LIN {X 0,Y 244.186,Z 1193.426,A -85,B 0,C 180,E1 11047.108,E2 11047.108} C_VEL
LIN {X 0,Y 247.926,Z 1188.555,A -85,B 0,C 180,E1 11042.035,E2 11042.035} C_VEL
LIN {X 0,Y 253.238,Z 1182.464,A -85,B 0,C 180,E1 11036.985,E2 11036.985} C_VEL
LIN {X 0,Y 261.489,Z 1173.839,A -85,B 0,C 180,E1 11031.267,E2 11031.267} C_VEL
LIN {X 0,Y 272.19,Z 1162.996,A -85,B 0,C 180,E1 11025.738,E2 11025.738} C_VEL
LIN {X 0,Y 282.22,Z 1152.992,A -85,B 0,C 180,E1 11021.623,E2 11021.623} C_VEL
LIN {X 0,Y 292.95,Z 1142.22,A -85,B 0,C 180,E1 11017.962,E2 11017.962} C_VEL
LIN {X 0,Y 305.97,Z 1128.885,A -85,B 0,C 180,E1 11014.233,E2 11014.233} C_VEL
LIN {X 0,Y 321.47,Z 1112.193,A -85,B 0,C 180,E1 11010.51,E2 11010.51} C_VEL
LIN {X 0,Y 333.886,Z 1098.086,A -85,B 0,C 180,E1 11007.944,E2 11007.944} C_VEL
LIN {X 0,Y 346.355,Z 1083.139,A -85,B 0,C 180,E1 11005.66,E2 11005.66} C_VEL
LIN {X 0,Y 358.973,Z 1067.071,A -85,B 0,C 180,E1 11003.599,E2 11003.599} C_VEL
LIN {X 0,Y 373.818,Z 1046.804,A -85,B 0,C 180,E1 11001.44,E2 11001.44} C_VEL
LIN {X 0,Y 387.51,Z 1026.01,A -85,B 0,C 180,E1 10999.648,E2 10999.648} C_VEL
LIN {X 0,Y 398.233,Z 1008.33,A -85,B 0,C 180,E1 10998.367,E2 10998.367} C_VEL
LIN {X 0,Y 408.718,Z 989.45,A -85,B 0,C 180,E1 10997.198,E2 10997.198} C_VEL
LIN {X 0,Y 418.525,Z 970.023,A -85,B 0,C 180,E1 10996.183,E2 10996.183} C_VEL
LIN {X 0,Y 429.683,Z 945.282,A -85,B 0,C 180,E1 10995.107,E2 10995.107} C_VEL
LIN {X 0,Y 439.012,Z 920.891,A -85,B 0,C 180,E1 10994.259,E2 10994.259} C_VEL
LIN {X 0,Y 446.039,Z 899.719,A -85,B 0,C 180,E1 10993.652,E2 10993.652} C_VEL
LIN {X 0,Y 452.043,Z 878.579,A -85,B 0,C 180,E1 10993.156,E2 10993.156} C_VEL
LIN {X 0,Y 457.537,Z 855.248,A -85,B 0,C 180,E1 10992.719,E2 10992.719} C_VEL
LIN {X 0,Y 462.73,Z 825.262,A -85,B 0,C 180,E1 10992.246,E2 10992.246} C_VEL
LIN {X 0,Y 469.946,Z 760.985,A -85,B 0,C 180,E1 10991.336,E2 10991.336} C_VEL
LIN {X 0,Y 484.421,Z 628.606,A -85,B 0,C 180,E1 10989.475,E2 10989.475} C_VEL
LIN {X 0,Y 483.133,Z 625.534,A -85,B 0,C 180,E1 10987.253,E2 10987.253} C_VEL
LIN {X 0,Y 482.186,Z 624.109,A -85,B 0,C 180,E1 10983.329,E2 10983.329} C_VEL
LIN {X 0,Y 483.259,Z 625.73,A -85,B 0,C 180,E1 10979.289,E2 10979.289} C_VEL
LIN {X 0,Y 484.397,Z 628.699,A -85,B 0,C 180,E1 10977.334,E2 10977.334} C_VEL
LIN {X 0,Y 463.189,Z 821.007,A -85,B 0,C 180,E1 10974.653,E2 10974.653} C_VEL
LIN {X 0,Y 459.068,Z 846.715,A -85,B 0,C 180,E1 10974.257,E2 10974.257} C_VEL
LIN {X 0,Y 452.825,Z 874.436,A -85,B 0,C 180,E1 10973.737,E2 10973.737} C_VEL
LIN {X 0,Y 446.811,Z 895.996,A -85,B 0,C 180,E1 10973.219,E2 10973.219} C_VEL
LIN {X 0,Y 440.078,Z 916.575,A -85,B 0,C 180,E1 10972.625,E2 10972.625} C_VEL
LIN {X 0,Y 432.249,Z 937.422,A -85,B 0,C 180,E1 10971.901,E2 10971.901} C_VEL
LIN {X 0,Y 421.642,Z 962.183,A -85,B 0,C 180,E1 10970.858,E2 10970.858} C_VEL
LIN {X 0,Y 410.101,Z 985.308,A -85,B 0,C 180,E1 10969.661,E2 10969.661} C_VEL
LIN {X 0,Y 399.598,Z 1004.318,A -85,B 0,C 180,E1 10968.484,E2 10968.484} C_VEL
LIN {X 0,Y 389.268,Z 1021.457,A -85,B 0,C 180,E1 10967.238,E2 10967.238} C_VEL
LIN {X 0,Y 377.601,Z 1039.273,A -85,B 0,C 180,E1 10965.728,E2 10965.728} C_VEL
LIN {X 0,Y 362.336,Z 1060.663,A -85,B 0,C 180,E1 10963.535,E2 10963.535} C_VEL
LIN {X 0,Y 348.036,Z 1078.861,A -85,B 0,C 180,E1 10961.23,E2 10961.23} C_VEL
LIN {X 0,Y 335.753,Z 1093.533,A -85,B 0,C 180,E1 10959.001,E2 10959.001} C_VEL
LIN {X 0,Y 322.991,Z 1107.947,A -85,B 0,C 180,E1 10956.391,E2 10956.391} C_VEL
LIN {X 0,Y 307.961,Z 1124.093,A -85,B 0,C 180,E1 10952.822,E2 10952.822} C_VEL
LIN {X 0,Y 293.963,Z 1138.215,A -85,B 0,C 180,E1 10948.868,E2 10948.868} C_VEL
LIN {X 0,Y 283.38,Z 1148.666,A -85,B 0,C 180,E1 10945.295,E2 10945.295} C_VEL
LIN {X 0,Y 273.45,Z 1158.351,A -85,B 0,C 180,E1 10941.297,E2 10941.297} C_VEL
LIN {X 0,Y 262.614,Z 1169.074,A -85,B 0,C 180,E1 10935.832,E2 10935.832} C_VEL
LIN {X 0,Y 253.878,Z 1177.853,A -85,B 0,C 180,E1 10929.937,E2 10929.937} C_VEL
LIN {X 0,Y 248.405,Z 1183.851,A -85,B 0,C 180,E1 10924.859,E2 10924.859} C_VEL
LIN {X 0,Y 244.451,Z 1188.7,A -85,B 0,C 180,E1 10919.664,E2 10919.664} C_VEL
LIN {X 0,Y 241.833,Z 1192.6,A -85,B 0,C 180,E1 10914.162,E2 10914.162} C_VEL
LIN {X 0,Y 240.342,Z 1195.722,A -85,B 0,C 180,E1 10907.679,E2 10907.679} C_VEL
LIN {X 0,Y 239.958,Z 1197.055,A -85,B 0,C 180,E1 10902.025,E2 10902.025} C_VEL
LIN {X 0,Y 239.922,Z 1197.274,A -85,B 0,C 180,E1 10897.182,E2 10897.182} C_VEL
LIN {X 0,Y 239.937,Z 1196.596,A -85,B 0,C 180,E1 10892.388,E2 10892.388} C_VEL
LIN {X 0,Y 240.18,Z 1194.92,A -85,B 0,C 180,E1 10887.375,E2 10887.375} C_VEL
LIN {X 0,Y 240.959,Z 1192.268,A -85,B 0,C 180,E1 10882.37,E2 10882.37} C_VEL
LIN {X 0,Y 242.622,Z 1188.623,A -85,B 0,C 180,E1 10877.384,E2 10877.384} C_VEL
LIN {X 0,Y 245.393,Z 1183.965,A -85,B 0,C 180,E1 10872.452,E2 10872.452} C_VEL
LIN {X 0,Y 249.359,Z 1178.262,A -85,B 0,C 180,E1 10867.609,E2 10867.609} C_VEL
LIN {X 0,Y 254.917,Z 1171.132,A -85,B 0,C 180,E1 10862.684,E2 10862.684} C_VEL
LIN {X 0,Y 263.638,Z 1160.802,A -85,B 0,C 180,E1 10856.949,E2 10856.949} C_VEL
LIN {X 0,Y 273.258,Z 1149.593,A -85,B 0,C 180,E1 10852.069,E2 10852.069} C_VEL
LIN {X 0,Y 282.441,Z 1139.053,A -85,B 0,C 180,E1 10848.277,E2 10848.277} C_VEL
LIN {X 0,Y 292.662,Z 1127.21,A -85,B 0,C 180,E1 10844.715,E2 10844.715} C_VEL
LIN {X 0,Y 305.879,Z 1111.538,A -85,B 0,C 180,E1 10840.828,E2 10840.828} C_VEL
LIN {X 0,Y 318.998,Z 1094.953,A -85,B 0,C 180,E1 10837.534,E2 10837.534} C_VEL
LIN {X 0,Y 330.002,Z 1080.382,A -85,B 0,C 180,E1 10835.109,E2 10835.109} C_VEL
LIN {X 0,Y 341.178,Z 1064.746,A -85,B 0,C 180,E1 10832.9,E2 10832.9} C_VEL
LIN {X 0,Y 353.523,Z 1046.342,A -85,B 0,C 180,E1 10830.707,E2 10830.707} C_VEL
LIN {X 0,Y 367.066,Z 1024.216,A -85,B 0,C 180,E1 10828.543,E2 10828.543} C_VEL
LIN {X 0,Y 377.623,Z 1005.303,A -85,B 0,C 180,E1 10827.005,E2 10827.005} C_VEL
LIN {X 0,Y 386.922,Z 987.177,A -85,B 0,C 180,E1 10825.75,E2 10825.75} C_VEL
LIN {X 0,Y 395.882,Z 967.953,A -85,B 0,C 180,E1 10824.601,E2 10824.601} C_VEL
LIN {X 0,Y 405.863,Z 944.175,A -85,B 0,C 180,E1 10823.413,E2 10823.413} C_VEL
LIN {X 0,Y 414.8,Z 919.187,A -85,B 0,C 180,E1 10822.403,E2 10822.403} C_VEL
LIN {X 0,Y 421.3,Z 898.161,A -85,B 0,C 180,E1 10821.7,E2 10821.7} C_VEL
LIN {X 0,Y 427.003,Z 876.597,A -85,B 0,C 180,E1 10821.107,E2 10821.107} C_VEL
LIN {X 0,Y 431.946,Z 854.086,A -85,B 0,C 180,E1 10820.608,E2 10820.608} C_VEL
LIN {X 0,Y 436.815,Z 824.39,A -85,B 0,C 180,E1 10820.087,E2 10820.087} C_VEL
LIN {X 0,Y 442.338,Z 770.319,A -85,B 0,C 180,E1 10819.277,E2 10819.277} C_VEL
LIN {X 0,Y 443.071,Z 762.736,A -85,B 0,C 180,E1 10819.166,E2 10819.166} C_VEL
LIN {X 0,Y 443.54,Z 755.2,A -85,B 0,C 180,E1 10818.932,E2 10818.932} C_VEL
LIN {X 0,Y 443.88,Z 735.631,A -85,B 0,C 180,E1 10817.865,E2 10817.865} C_VEL
LIN {X 0,Y 444.333,Z 729.152,A -85,B 0,C 180,E1 10817.674,E2 10817.674} C_VEL
LIN {X 0,Y 455.797,Z 614.554,A -85,B 0,C 180,E1 10816.017,E2 10816.017} C_VEL
LIN {X 0,Y 452.593,Z 608.182,A -85,B 0,C 180,E1 10813.413,E2 10813.413} C_VEL
LIN {X 0,Y 449.906,Z 603.038,A -85,B 0,C 180,E1 10810.5,E2 10810.5} C_VEL
LIN {X 0,Y 448.146,Z 599.162,A -85,B 0,C 180,E1 10807.435,E2 10807.435} C_VEL
LIN {X 0,Y 447.268,Z 598.262,A -85,B 0,C 180,E1 10803.076,E2 10803.076} C_VEL
LIN {X 0,Y 448.281,Z 599.424,A -85,B 0,C 180,E1 10799.361,E2 10799.361} C_VEL
LIN {X 0,Y 450.497,Z 604.17,A -85,B 0,C 180,E1 10795.863,E2 10795.863} C_VEL
LIN {X 0,Y 452.759,Z 608.569,A -85,B 0,C 180,E1 10793.533,E2 10793.533} C_VEL
LIN {X 0,Y 455.853,Z 614.635,A -85,B 0,C 180,E1 10791.049,E2 10791.049} C_VEL
LIN {X 0,Y 435.182,Z 820.905,A -85,B 0,C 180,E1 10788.056,E2 10788.056} C_VEL
LIN {X 0,Y 431.958,Z 843.365,A -85,B 0,C 180,E1 10787.688,E2 10787.688} C_VEL
LIN {X 0,Y 426.641,Z 870.513,A -85,B 0,C 180,E1 10787.178,E2 10787.178} C_VEL
LIN {X 0,Y 419.824,Z 896.759,A -85,B 0,C 180,E1 10786.528,E2 10786.528} C_VEL
LIN {X 0,Y 413.42,Z 917.629,A -85,B 0,C 180,E1 10785.887,E2 10785.887} C_VEL
LIN {X 0,Y 406.063,Z 938.493,A -85,B 0,C 180,E1 10785.118,E2 10785.118} C_VEL
LIN {X 0,Y 397.094,Z 960.94,A -85,B 0,C 180,E1 10784.123,E2 10784.123} C_VEL
LIN {X 0,Y 385.324,Z 986.555,A -85,B 0,C 180,E1 10782.727,E2 10782.727} C_VEL
LIN {X 0,Y 375.033,Z 1006.507,A -85,B 0,C 180,E1 10781.41,E2 10781.41} C_VEL
LIN {X 0,Y 364.937,Z 1024.459,A -85,B 0,C 180,E1 10780.01,E2 10780.01} C_VEL
LIN {X 0,Y 353.893,Z 1042.554,A -85,B 0,C 180,E1 10778.361,E2 10778.361} C_VEL
LIN {X 0,Y 339.406,Z 1064.376,A -85,B 0,C 180,E1 10775.955,E2 10775.955} C_VEL
LIN {X 0,Y 326.96,Z 1081.567,A -85,B 0,C 180,E1 10773.637,E2 10773.637} C_VEL
LIN {X 0,Y 315.749,Z 1096.194,A -85,B 0,C 180,E1 10771.3,E2 10771.3} C_VEL
LIN {X 0,Y 304.43,Z 1110.258,A -85,B 0,C 180,E1 10768.642,E2 10768.642} C_VEL
LIN {X 0,Y 292.495,Z 1124.488,A -85,B 0,C 180,E1 10765.426,E2 10765.426} C_VEL
LIN {X 0,Y 278.355,Z 1140.667,A -85,B 0,C 180,E1 10760.884,E2 10760.884} C_VEL
LIN {X 0,Y 268.219,Z 1151.989,A -85,B 0,C 180,E1 10756.94,E2 10756.94} C_VEL
LIN {X 0,Y 259.27,Z 1161.988,A -85,B 0,C 180,E1 10752.744,E2 10752.744} C_VEL
LIN {X 0,Y 251.084,Z 1171.395,A -85,B 0,C 180,E1 10747.955,E2 10747.955} C_VEL
LIN {X 0,Y 242.869,Z 1181.4,A -85,B 0,C 180,E1 10741.523,E2 10741.523} C_VEL
LIN {X 0,Y 237.906,Z 1188.149,A -85,B 0,C 180,E1 10735.918,E2 10735.918} C_VEL
LIN {X 0,Y 234.944,Z 1192.933,A -85,B 0,C 180,E1 10730.945,E2 10730.945} C_VEL
LIN {X 0,Y 233.123,Z 1196.719,A -85,B 0,C 180,E1 10725.932,E2 10725.932} C_VEL
LIN {X 0,Y 232.218,Z 1199.53,A -85,B 0,C 180,E1 10720.921,E2 10720.921} C_VEL
LIN {X 0,Y 231.957,Z 1201.252,A -85,B 0,C 180,E1 10716.435,E2 10716.435} C_VEL
LIN {X 0,Y 231.917,Z 1202.222,A -85,B 0,C 180,E1 10711.976,E2 10711.976} C_VEL
LIN {X 0,Y 231.915,Z 1202.429,A -85,B 0,C 180,E1 10707.282,E2 10707.282} C_VEL
LIN {X 0,Y 232.002,Z 1201.743,A -85,B 0,C 180,E1 10702.322,E2 10702.322} C_VEL
LIN {X 0,Y 232.542,Z 1199.921,A -85,B 0,C 180,E1 10696.828,E2 10696.828} C_VEL
LIN {X 0,Y 233.985,Z 1197.172,A -85,B 0,C 180,E1 10691.564,E2 10691.564} C_VEL
LIN {X 0,Y 236.752,Z 1193.212,A -85,B 0,C 180,E1 10686.082,E2 10686.082} C_VEL
LIN {X 0,Y 240.774,Z 1188.384,A -85,B 0,C 180,E1 10680.931,E2 10680.931} C_VEL
LIN {X 0,Y 246.574,Z 1182.199,A -85,B 0,C 180,E1 10675.692,E2 10675.692} C_VEL
LIN {X 0,Y 255.93,Z 1173.039,A -85,B 0,C 180,E1 10669.57,E2 10669.57} C_VEL
LIN {X 0,Y 266.962,Z 1162.4,A -85,B 0,C 180,E1 10664.159,E2 10664.159} C_VEL
LIN {X 0,Y 277.257,Z 1152.614,A -85,B 0,C 180,E1 10660.135,E2 10660.135} C_VEL
LIN {X 0,Y 288.471,Z 1141.814,A -85,B 0,C 180,E1 10656.474,E2 10656.474} C_VEL
LIN {X 0,Y 303.298,Z 1127.191,A -85,B 0,C 180,E1 10652.442,E2 10652.442} C_VEL
LIN {X 0,Y 318.724,Z 1110.926,A -85,B 0,C 180,E1 10648.927,E2 10648.927} C_VEL
LIN {X 0,Y 331.554,Z 1096.708,A -85,B 0,C 180,E1 10646.408,E2 10646.408} C_VEL
LIN {X 0,Y 344.207,Z 1081.859,A -85,B 0,C 180,E1 10644.201,E2 10644.201} C_VEL
LIN {X 0,Y 358.922,Z 1063.45,A -85,B 0,C 180,E1 10641.929,E2 10641.929} C_VEL
LIN {X 0,Y 374.154,Z 1042.484,A -85,B 0,C 180,E1 10639.839,E2 10639.839} C_VEL
LIN {X 0,Y 386.517,Z 1023.899,A -85,B 0,C 180,E1 10638.31,E2 10638.31} C_VEL
LIN {X 0,Y 397.46,Z 1006.022,A -85,B 0,C 180,E1 10637.073,E2 10637.073} C_VEL
LIN {X 0,Y 408.18,Z 986.828,A -85,B 0,C 180,E1 10635.936,E2 10635.936} C_VEL
LIN {X 0,Y 420.416,Z 962.429,A -85,B 0,C 180,E1 10634.743,E2 10634.743} C_VEL
LIN {X 0,Y 430.416,Z 939.336,A -85,B 0,C 180,E1 10633.829,E2 10633.829} C_VEL
LIN {X 0,Y 438.081,Z 919.278,A -85,B 0,C 180,E1 10633.169,E2 10633.169} C_VEL
LIN {X 0,Y 444.945,Z 898.704,A -85,B 0,C 180,E1 10632.604,E2 10632.604} C_VEL
LIN {X 0,Y 451.113,Z 877.071,A -85,B 0,C 180,E1 10632.118,E2 10632.118} C_VEL
LIN {X 0,Y 457.429,Z 849.933,A -85,B 0,C 180,E1 10631.636,E2 10631.636} C_VEL
LIN {X 0,Y 461.849,Z 822.889,A -85,B 0,C 180,E1 10631.226,E2 10631.226} C_VEL
LIN {X 0,Y 479.309,Z 667.042,A -85,B 0,C 180,E1 10629.077,E2 10629.077} C_VEL
LIN {X 0,Y 482.848,Z 635.475,A -85,B 0,C 180,E1 10628.635,E2 10628.635} C_VEL
LIN {X 0,Y 482.041,Z 633.376,A -85,B 0,C 180,E1 10627.03,E2 10627.03} C_VEL
LIN {X 0,Y 481.209,Z 632.051,A -85,B 0,C 180,E1 10623.335,E2 10623.335} C_VEL
LIN {X 0,Y 482.215,Z 633.613,A -85,B 0,C 180,E1 10619.406,E2 10619.406} C_VEL
LIN {X 0,Y 482.811,Z 635.606,A -85,B 0,C 180,E1 10618.188,E2 10618.188} C_VEL
LIN {X 0,Y 461.996,Z 821.153,A -85,B 0,C 180,E1 10615.636,E2 10615.636} C_VEL
LIN {X 0,Y 457.786,Z 847.04,A -85,B 0,C 180,E1 10615.245,E2 10615.245} C_VEL
LIN {X 0,Y 451.491,Z 874.603,A -85,B 0,C 180,E1 10614.741,E2 10614.741} C_VEL
LIN {X 0,Y 445.434,Z 896.052,A -85,B 0,C 180,E1 10614.24,E2 10614.24} C_VEL
LIN {X 0,Y 438.617,Z 916.629,A -85,B 0,C 180,E1 10613.663,E2 10613.663} C_VEL
LIN {X 0,Y 430.895,Z 936.94,A -85,B 0,C 180,E1 10612.978,E2 10612.978} C_VEL
LIN {X 0,Y 420.529,Z 960.923,A -85,B 0,C 180,E1 10612.003,E2 10612.003} C_VEL
LIN {X 0,Y 408.715,Z 984.431,A -85,B 0,C 180,E1 10610.829,E2 10610.829} C_VEL
LIN {X 0,Y 397.896,Z 1003.772,A -85,B 0,C 180,E1 10609.667,E2 10609.667} C_VEL
LIN {X 0,Y 387.294,Z 1021.09,A -85,B 0,C 180,E1 10608.445,E2 10608.445} C_VEL
LIN {X 0,Y 375.232,Z 1039.194,A -85,B 0,C 180,E1 10606.948,E2 10606.948} C_VEL
LIN {X 0,Y 360.165,Z 1059.97,A -85,B 0,C 180,E1 10604.873,E2 10604.873} C_VEL
LIN {X 0,Y 345.292,Z 1078.493,A -85,B 0,C 180,E1 10602.578,E2 10602.578} C_VEL
LIN {X 0,Y 332.361,Z 1093.574,A -85,B 0,C 180,E1 10600.324,E2 10600.324} C_VEL
LIN {X 0,Y 319.126,Z 1108.112,A -85,B 0,C 180,E1 10597.721,E2 10597.721} C_VEL
LIN {X 0,Y 303.385,Z 1124.464,A -85,B 0,C 180,E1 10594.121,E2 10594.121} C_VEL
LIN {X 0,Y 289.734,Z 1137.77,A -85,B 0,C 180,E1 10590.416,E2 10590.416} C_VEL
LIN {X 0,Y 278.471,Z 1148.451,A -85,B 0,C 180,E1 10586.782,E2 10586.782} C_VEL
LIN {X 0,Y 267.829,Z 1158.373,A -85,B 0,C 180,E1 10582.671,E2 10582.671} C_VEL
LIN {X 0,Y 256.793,Z 1168.725,A -85,B 0,C 180,E1 10577.35,E2 10577.35} C_VEL
LIN {X 0,Y 247.261,Z 1177.764,A -85,B 0,C 180,E1 10571.233,E2 10571.233} C_VEL
LIN {X 0,Y 241.35,Z 1183.79,A -85,B 0,C 180,E1 10566.035,E2 10566.035} C_VEL
LIN {X 0,Y 237.211,Z 1188.459,A -85,B 0,C 180,E1 10560.946,E2 10560.946} C_VEL
LIN {X 0,Y 234.434,Z 1192.114,A -85,B 0,C 180,E1 10555.787,E2 10555.787} C_VEL
LIN {X 0,Y 232.81,Z 1194.814,A -85,B 0,C 180,E1 10550.562,E2 10550.562} C_VEL
LIN {X 0,Y 232.131,Z 1196.512,A -85,B 0,C 180,E1 10545.489,E2 10545.489} C_VEL
LIN {X 0,Y 231.939,Z 1197.262,A -85,B 0,C 180,E1 10540.934,E2 10540.934} C_VEL
LIN {X 0,Y 231.922,Z 1197.305,A -85,B 0,C 180,E1 10536.685,E2 10536.685} C_VEL
LIN {X 0,Y 231.945,Z 1196.588,A -85,B 0,C 180,E1 10531.976,E2 10531.976} C_VEL
LIN {X 0,Y 232.21,Z 1194.962,A -85,B 0,C 180,E1 10527.038,E2 10527.038} C_VEL
LIN {X 0,Y 233.075,Z 1192.291,A -85,B 0,C 180,E1 10521.862,E2 10521.862} C_VEL
LIN {X 0,Y 234.893,Z 1188.628,A -85,B 0,C 180,E1 10516.711,E2 10516.711} C_VEL
LIN {X 0,Y 237.87,Z 1183.95,A -85,B 0,C 180,E1 10511.624,E2 10511.624} C_VEL
LIN {X 0,Y 242.127,Z 1178.229,A -85,B 0,C 180,E1 10506.645,E2 10506.645} C_VEL
LIN {X 0,Y 248.032,Z 1171.08,A -85,B 0,C 180,E1 10501.597,E2 10501.597} C_VEL
LIN {X 0,Y 257.321,Z 1160.616,A -85,B 0,C 180,E1 10495.708,E2 10495.708} C_VEL
LIN {X 0,Y 267.344,Z 1149.472,A -85,B 0,C 180,E1 10490.798,E2 10490.798} C_VEL
LIN {X 0,Y 276.941,Z 1138.906,A -85,B 0,C 180,E1 10486.972,E2 10486.972} C_VEL
LIN {X 0,Y 287.569,Z 1127.032,A -85,B 0,C 180,E1 10483.392,E2 10483.392} C_VEL
LIN {X 0,Y 300.955,Z 1111.667,A -85,B 0,C 180,E1 10479.577,E2 10479.577} C_VEL
LIN {X 0,Y 314.811,Z 1094.65,A -85,B 0,C 180,E1 10476.212,E2 10476.212} C_VEL
LIN {X 0,Y 326.114,Z 1080.069,A -85,B 0,C 180,E1 10473.811,E2 10473.811} C_VEL
LIN {X 0,Y 337.668,Z 1064.282,A -85,B 0,C 180,E1 10471.61,E2 10471.61} C_VEL
LIN {X 0,Y 351.72,Z 1043.749,A -85,B 0,C 180,E1 10469.223,E2 10469.223} C_VEL
LIN {X 0,Y 364.462,Z 1023.05,A -85,B 0,C 180,E1 10467.269,E2 10467.269} C_VEL
LIN {X 0,Y 374.845,Z 1004.734,A -85,B 0,C 180,E1 10465.81,E2 10465.81} C_VEL
LIN {X 0,Y 384.68,Z 985.823,A -85,B 0,C 180,E1 10464.534,E2 10464.534} C_VEL
LIN {X 0,Y 394.662,Z 964.588,A -85,B 0,C 180,E1 10463.31,E2 10463.31} C_VEL
LIN {X 0,Y 405.233,Z 938.926,A -85,B 0,C 180,E1 10462.106,E2 10462.106} C_VEL
LIN {X 0,Y 413.051,Z 916.965,A -85,B 0,C 180,E1 10461.259,E2 10461.259} C_VEL
LIN {X 0,Y 419.421,Z 896.418,A -85,B 0,C 180,E1 10460.6,E2 10460.6} C_VEL
LIN {X 0,Y 425.335,Z 874.042,A -85,B 0,C 180,E1 10460.009,E2 10460.009} C_VEL
LIN {X 0,Y 431.234,Z 846.296,A -85,B 0,C 180,E1 10459.436,E2 10459.436} C_VEL
LIN {X 0,Y 435.083,Z 820.686,A -85,B 0,C 180,E1 10459.013,E2 10459.013} C_VEL
LIN {X 0,Y 444.333,Z 729.152,A -85,B 0,C 180,E1 10457.674,E2 10457.674} C_VEL
LIN {X 0,Y 444.838,Z 721.621,A -85,B 0,C 180,E1 10457.437,E2 10457.437} C_VEL
LIN {X 0,Y 445.38,Z 702.061,A -85,B 0,C 180,E1 10456.371,E2 10456.371} C_VEL
LIN {X 0,Y 445.875,Z 695.582,A -85,B 0,C 180,E1 10456.184,E2 10456.184} C_VEL
LIN {X 0,Y 453.534,Z 620.483,A -85,B 0,C 180,E1 10455.099,E2 10455.099} C_VEL
LIN {X 0,Y 450.948,Z 615.057,A -85,B 0,C 180,E1 10452.811,E2 10452.811} C_VEL
LIN {X 0,Y 448.733,Z 610.783,A -85,B 0,C 180,E1 10450.269,E2 10450.269} C_VEL
LIN {X 0,Y 447.113,Z 607.072,A -85,B 0,C 180,E1 10447.324,E2 10447.324} C_VEL
LIN {X 0,Y 446.298,Z 606.204,A -85,B 0,C 180,E1 10442.954,E2 10442.954} C_VEL
LIN {X 0,Y 447.238,Z 607.309,A -85,B 0,C 180,E1 10439.488,E2 10439.488} C_VEL
LIN {X 0,Y 449.343,Z 611.965,A -85,B 0,C 180,E1 10436.044,E2 10436.044} C_VEL
LIN {X 0,Y 451.479,Z 616.243,A -85,B 0,C 180,E1 10433.77,E2 10433.77} C_VEL
LIN {X 0,Y 453.589,Z 620.717,A -85,B 0,C 180,E1 10431.952,E2 10431.952} C_VEL
LIN {X 0,Y 432.917,Z 822.739,A -85,B 0,C 180,E1 10429.052,E2 10429.052} C_VEL
LIN {X 0,Y 429.15,Z 847.665,A -85,B 0,C 180,E1 10428.646,E2 10428.646} C_VEL
LIN {X 0,Y 423.012,Z 876.287,A -85,B 0,C 180,E1 10428.091,E2 10428.091} C_VEL
LIN {X 0,Y 417.089,Z 898.368,A -85,B 0,C 180,E1 10427.54,E2 10427.54} C_VEL
LIN {X 0,Y 410.566,Z 919.112,A -85,B 0,C 180,E1 10426.909,E2 10426.909} C_VEL
LIN {X 0,Y 402.712,Z 940.838,A -85,B 0,C 180,E1 10426.114,E2 10426.114} C_VEL
LIN {X 0,Y 391.464,Z 967.728,A -85,B 0,C 180,E1 10424.898,E2 10424.898} C_VEL
LIN {X 0,Y 381.668,Z 988.217,A -85,B 0,C 180,E1 10423.764,E2 10423.764} C_VEL
LIN {X 0,Y 371.79,Z 1006.964,A -85,B 0,C 180,E1 10422.539,E2 10422.539} C_VEL
LIN {X 0,Y 361.85,Z 1024.288,A -85,B 0,C 180,E1 10421.21,E2 10421.21} C_VEL
LIN {X 0,Y 350.489,Z 1042.531,A -85,B 0,C 180,E1 10419.574,E2 10419.574} C_VEL
LIN {X 0,Y 335.301,Z 1064.865,A -85,B 0,C 180,E1 10417.135,E2 10417.135} C_VEL
LIN {X 0,Y 322.569,Z 1082.009,A -85,B 0,C 180,E1 10414.837,E2 10414.837} C_VEL
LIN {X 0,Y 311.079,Z 1096.589,A -85,B 0,C 180,E1 10412.512,E2 10412.512} C_VEL
LIN {X 0,Y 299.451,Z 1110.61,A -85,B 0,C 180,E1 10409.859,E2 10409.859} C_VEL
LIN {X 0,Y 286.001,Z 1126.151,A -85,B 0,C 180,E1 10406.309,E2 10406.309} C_VEL
LIN {X 0,Y 272.532,Z 1140.91,A -85,B 0,C 180,E1 10402.072,E2 10402.072} C_VEL
LIN {X 0,Y 262.019,Z 1152.2,A -85,B 0,C 180,E1 10398.083,E2 10398.083} C_VEL
LIN {X 0,Y 252.7,Z 1162.17,A -85,B 0,C 180,E1 10393.822,E2 10393.822} C_VEL
LIN {X 0,Y 243.971,Z 1171.731,A -85,B 0,C 180,E1 10388.832,E2 10388.832} C_VEL
LIN {X 0,Y 235.494,Z 1181.5,A -85,B 0,C 180,E1 10382.334,E2 10382.334} C_VEL
LIN {X 0,Y 230.455,Z 1187.953,A -85,B 0,C 180,E1 10376.822,E2 10376.822} C_VEL
LIN {X 0,Y 227.249,Z 1192.759,A -85,B 0,C 180,E1 10371.69,E2 10371.69} C_VEL
LIN {X 0,Y 225.261,Z 1196.565,A -85,B 0,C 180,E1 10366.503,E2 10366.503} C_VEL
LIN {X 0,Y 224.256,Z 1199.396,A -85,B 0,C 180,E1 10361.313,E2 10361.313} C_VEL
LIN {X 0,Y 223.963,Z 1201.137,A -85,B 0,C 180,E1 10356.666,E2 10356.666} C_VEL
LIN {X 0,Y 223.917,Z 1202.126,A -85,B 0,C 180,E1 10352.047,E2 10352.047} C_VEL
LIN {X 0,Y 223.915,Z 1202.35,A -85,B 0,C 180,E1 10347.185,E2 10347.185} C_VEL
LIN {X 0,Y 224.021,Z 1201.612,A -85,B 0,C 180,E1 10341.789,E2 10341.789} C_VEL
LIN {X 0,Y 224.623,Z 1199.877,A -85,B 0,C 180,E1 10336.354,E2 10336.354} C_VEL
LIN {X 0,Y 226.199,Z 1197.148,A -85,B 0,C 180,E1 10330.907,E2 10330.907} C_VEL
LIN {X 0,Y 229.209,Z 1193.207,A -85,B 0,C 180,E1 10325.243,E2 10325.243} C_VEL
LIN {X 0,Y 233.666,Z 1188.271,A -85,B 0,C 180,E1 10319.813,E2 10319.813} C_VEL
LIN {X 0,Y 239.721,Z 1182.235,A -85,B 0,C 180,E1 10314.566,E2 10314.566} C_VEL
LIN {X 0,Y 249.203,Z 1173.48,A -85,B 0,C 180,E1 10308.546,E2 10308.546} C_VEL
LIN {X 0,Y 260.917,Z 1162.756,A -85,B 0,C 180,E1 10302.952,E2 10302.952} C_VEL
LIN {X 0,Y 271.937,Z 1152.749,A -85,B 0,C 180,E1 10298.787,E2 10298.787} C_VEL
LIN {X 0,Y 283.843,Z 1141.738,A -85,B 0,C 180,E1 10295.044,E2 10295.044} C_VEL
LIN {X 0,Y 298.912,Z 1127.384,A -85,B 0,C 180,E1 10291.095,E2 10291.095} C_VEL
LIN {X 0,Y 314.793,Z 1111.181,A -85,B 0,C 180,E1 10287.604,E2 10287.604} C_VEL
LIN {X 0,Y 327.963,Z 1096.996,A -85,B 0,C 180,E1 10285.115,E2 10285.115} C_VEL
LIN {X 0,Y 340.703,Z 1082.441,A -85,B 0,C 180,E1 10282.975,E2 10282.975} C_VEL
LIN {X 0,Y 354.333,Z 1065.812,A -85,B 0,C 180,E1 10280.931,E2 10280.931} C_VEL
LIN {X 0,Y 371.159,Z 1043.4,A -85,B 0,C 180,E1 10278.698,E2 10278.698} C_VEL
LIN {X 0,Y 384.048,Z 1024.418,A -85,B 0,C 180,E1 10277.163,E2 10277.163} C_VEL
LIN {X 0,Y 395.168,Z 1006.598,A -85,B 0,C 180,E1 10275.955,E2 10275.955} C_VEL
LIN {X 0,Y 405.567,Z 988.352,A -85,B 0,C 180,E1 10274.893,E2 10274.893} C_VEL
LIN {X 0,Y 416.118,Z 967.949,A -85,B 0,C 180,E1 10273.895,E2 10273.895} C_VEL
LIN {X 0,Y 428.138,Z 941.392,A -85,B 0,C 180,E1 10272.836,E2 10272.836} C_VEL
LIN {X 0,Y 436.684,Z 919.415,A -85,B 0,C 180,E1 10272.128,E2 10272.128} C_VEL
LIN {X 0,Y 443.793,Z 898.355,A -85,B 0,C 180,E1 10271.568,E2 10271.568} C_VEL
LIN {X 0,Y 450.039,Z 876.651,A -85,B 0,C 180,E1 10271.098,E2 10271.098} C_VEL
LIN {X 0,Y 456.422,Z 849.35,A -85,B 0,C 180,E1 10270.629,E2 10270.629} C_VEL
LIN {X 0,Y 460.811,Z 822.792,A -85,B 0,C 180,E1 10270.235,E2 10270.235} C_VEL
LIN {X 0,Y 478.798,Z 664.967,A -85,B 0,C 180,E1 10268.091,E2 10268.091} C_VEL
LIN {X 0,Y 481.382,Z 642.238,A -85,B 0,C 180,E1 10267.759,E2 10267.759} C_VEL
LIN {X 0,Y 480.956,Z 641.216,A -85,B 0,C 180,E1 10266.806,E2 10266.806} C_VEL
LIN {X 0,Y 480.233,Z 640.001,A -85,B 0,C 180,E1 10263.223,E2 10263.223} C_VEL
LIN {X 0,Y 481.173,Z 641.496,A -85,B 0,C 180,E1 10259.524,E2 10259.524} C_VEL
LIN {X 0,Y 481.351,Z 642.417,A -85,B 0,C 180,E1 10259.048,E2 10259.048} C_VEL
LIN {X 0,Y 460.939,Z 821.304,A -85,B 0,C 180,E1 10256.623,E2 10256.623} C_VEL
LIN {X 0,Y 456.643,Z 847.359,A -85,B 0,C 180,E1 10256.237,E2 10256.237} C_VEL
LIN {X 0,Y 450.276,Z 874.847,A -85,B 0,C 180,E1 10255.75,E2 10255.75} C_VEL
LIN {X 0,Y 444.2,Z 896.11,A -85,B 0,C 180,E1 10255.268,E2 10255.268} C_VEL
LIN {X 0,Y 437.301,Z 916.687,A -85,B 0,C 180,E1 10254.707,E2 10254.707} C_VEL
LIN {X 0,Y 429.741,Z 936.359,A -85,B 0,C 180,E1 10254.065,E2 10254.065} C_VEL
LIN {X 0,Y 420.372,Z 957.872,A -85,B 0,C 180,E1 10253.228,E2 10253.228} C_VEL
LIN {X 0,Y 407.265,Z 983.989,A -85,B 0,C 180,E1 10251.981,E2 10251.981} C_VEL
LIN {X 0,Y 396.012,Z 1003.816,A -85,B 0,C 180,E1 10250.823,E2 10250.823} C_VEL
LIN {X 0,Y 385.232,Z 1021.134,A -85,B 0,C 180,E1 10249.634,E2 10249.634} C_VEL
LIN {X 0,Y 372.878,Z 1039.35,A -85,B 0,C 180,E1 10248.162,E2 10248.162} C_VEL
LIN {X 0,Y 357.028,Z 1060.709,A -85,B 0,C 180,E1 10246.063,E2 10246.063} C_VEL
LIN {X 0,Y 341.988,Z 1079.014,A -85,B 0,C 180,E1 10243.826,E2 10243.826} C_VEL
LIN {X 0,Y 329.018,Z 1093.762,A -85,B 0,C 180,E1 10241.65,E2 10241.65} C_VEL
LIN {X 0,Y 316.381,Z 1107.289,A -85,B 0,C 180,E1 10239.27,E2 10239.27} C_VEL
LIN {X 0,Y 301.792,Z 1122.079,A -85,B 0,C 180,E1 10236.121,E2 10236.121} C_VEL
LIN {X 0,Y 285.512,Z 1137.526,A -85,B 0,C 180,E1 10231.945,E2 10231.945} C_VEL
LIN {X 0,Y 273.512,Z 1148.462,A -85,B 0,C 180,E1 10228.235,E2 10228.235} C_VEL
LIN {X 0,Y 262.588,Z 1158.192,A -85,B 0,C 180,E1 10224.198,E2 10224.198} C_VEL
LIN {X 0,Y 251.876,Z 1167.709,A -85,B 0,C 180,E1 10219.306,E2 10219.306} C_VEL
LIN {X 0,Y 240.953,Z 1177.51,A -85,B 0,C 180,E1 10212.734,E2 10212.734} C_VEL
LIN {X 0,Y 234.397,Z 1183.73,A -85,B 0,C 180,E1 10207.281,E2 10207.281} C_VEL
LIN {X 0,Y 229.815,Z 1188.497,A -85,B 0,C 180,E1 10201.96,E2 10201.96} C_VEL
LIN {X 0,Y 226.672,Z 1192.285,A -85,B 0,C 180,E1 10196.431,E2 10196.431} C_VEL
LIN {X 0,Y 224.896,Z 1194.977,A -85,B 0,C 180,E1 10190.986,E2 10190.986} C_VEL
LIN {X 0,Y 224.135,Z 1196.696,A -85,B 0,C 180,E1 10185.525,E2 10185.525} C_VEL
LIN {X 0,Y 223.937,Z 1197.403,A -85,B 0,C 180,E1 10180.548,E2 10180.548} C_VEL
LIN {X 0,Y 223.923,Z 1197.337,A -85,B 0,C 180,E1 10176.152,E2 10176.152} C_VEL
LIN {X 0,Y 223.948,Z 1196.647,A -85,B 0,C 180,E1 10171.791,E2 10171.791} C_VEL
LIN {X 0,Y 224.22,Z 1195.114,A -85,B 0,C 180,E1 10166.933,E2 10166.933} C_VEL
LIN {X 0,Y 225.138,Z 1192.47,A -85,B 0,C 180,E1 10161.573,E2 10161.573} C_VEL
LIN {X 0,Y 227.07,Z 1188.834,A -85,B 0,C 180,E1 10156.245,E2 10156.245} C_VEL
LIN {X 0,Y 230.22,Z 1184.184,A -85,B 0,C 180,E1 10150.99,E2 10150.99} C_VEL
LIN {X 0,Y 234.714,Z 1178.491,A -85,B 0,C 180,E1 10145.861,E2 10145.861} C_VEL
LIN {X 0,Y 240.919,Z 1171.369,A -85,B 0,C 180,E1 10140.678,E2 10140.678} C_VEL
LIN {X 0,Y 250.252,Z 1161.411,A -85,B 0,C 180,E1 10134.877,E2 10134.877} C_VEL
LIN {X 0,Y 261.24,Z 1149.7,A -85,B 0,C 180,E1 10129.612,E2 10129.612} C_VEL
LIN {X 0,Y 271.589,Z 1138.754,A -85,B 0,C 180,E1 10125.614,E2 10125.614} C_VEL
LIN {X 0,Y 283.133,Z 1126.318,A -85,B 0,C 180,E1 10121.871,E2 10121.871} C_VEL
LIN {X 0,Y 298.361,Z 1109.174,A -85,B 0,C 180,E1 10117.733,E2 10117.733} C_VEL
LIN {X 0,Y 310.74,Z 1094.407,A -85,B 0,C 180,E1 10114.865,E2 10114.865} C_VEL
LIN {X 0,Y 322.395,Z 1079.757,A -85,B 0,C 180,E1 10112.482,E2 10112.482} C_VEL
LIN {X 0,Y 334.169,Z 1064.039,A -85,B 0,C 180,E1 10110.321,E2 10110.321} C_VEL
LIN {X 0,Y 348.343,Z 1043.752,A -85,B 0,C 180,E1 10107.999,E2 10107.999} C_VEL
LIN {X 0,Y 361.255,Z 1023.202,A -85,B 0,C 180,E1 10106.087,E2 10106.087} C_VEL
LIN {X 0,Y 371.839,Z 1004.882,A -85,B 0,C 180,E1 10104.651,E2 10104.651} C_VEL
LIN {X 0,Y 381.445,Z 986.763,A -85,B 0,C 180,E1 10103.447,E2 10103.447} C_VEL
LIN {X 0,Y 390.769,Z 967.374,A -85,B 0,C 180,E1 10102.337,E2 10102.337} C_VEL
LIN {X 0,Y 401.458,Z 942.502,A -85,B 0,C 180,E1 10101.158,E2 10101.158} C_VEL
LIN {X 0,Y 410.258,Z 918.379,A -85,B 0,C 180,E1 10100.232,E2 10100.232} C_VEL
LIN {X 0,Y 416.802,Z 897.736,A -85,B 0,C 180,E1 10099.578,E2 10099.578} C_VEL
LIN {X 0,Y 422.574,Z 876.452,A -85,B 0,C 180,E1 10099.02,E2 10099.02} C_VEL
LIN {X 0,Y 427.716,Z 853.579,A -85,B 0,C 180,E1 10098.537,E2 10098.537} C_VEL
LIN {X 0,Y 432.716,Z 823.437,A -85,B 0,C 180,E1 10098.03,E2 10098.03} C_VEL
LIN {X 0,Y 439.264,Z 761.032,A -85,B 0,C 180,E1 10097.121,E2 10097.121} C_VEL
LIN {X 0,Y 445.875,Z 695.582,A -85,B 0,C 180,E1 10096.184,E2 10096.184} C_VEL
LIN {X 0,Y 446.428,Z 688.051,A -85,B 0,C 180,E1 10095.95,E2 10095.95} C_VEL
LIN {X 0,Y 447.174,Z 668.504,A -85,B 0,C 180,E1 10094.886,E2 10094.886} C_VEL
LIN {X 0,Y 447.703,Z 662.025,A -85,B 0,C 180,E1 10094.701,E2 10094.701} C_VEL
LIN {X 0,Y 451.418,Z 626.427,A -85,B 0,C 180,E1 10094.2,E2 10094.2} C_VEL
LIN {X 0,Y 449.327,Z 622.157,A -85,B 0,C 180,E1 10092.205,E2 10092.205} C_VEL
LIN {X 0,Y 447.568,Z 618.528,A -85,B 0,C 180,E1 10090.035,E2 10090.035} C_VEL
LIN {X 0,Y 446.081,Z 614.981,A -85,B 0,C 180,E1 10087.211,E2 10087.211} C_VEL
LIN {X 0,Y 445.32,Z 614.146,A -85,B 0,C 180,E1 10082.96,E2 10082.96} C_VEL
LIN {X 0,Y 446.197,Z 615.192,A -85,B 0,C 180,E1 10079.615,E2 10079.615} C_VEL
LIN {X 0,Y 448.243,Z 619.88,A -85,B 0,C 180,E1 10076.163,E2 10076.163} C_VEL
LIN {X 0,Y 450.272,Z 624.059,A -85,B 0,C 180,E1 10073.945,E2 10073.945} C_VEL
LIN {X 0,Y 451.442,Z 626.65,A -85,B 0,C 180,E1 10072.867,E2 10072.867} C_VEL
LIN {X 0,Y 430.996,Z 822.835,A -85,B 0,C 180,E1 10070.084,E2 10070.084} C_VEL
LIN {X 0,Y 427.071,Z 848.325,A -85,B 0,C 180,E1 10069.676,E2 10069.676} C_VEL
LIN {X 0,Y 420.913,Z 876.475,A -85,B 0,C 180,E1 10069.142,E2 10069.142} C_VEL
LIN {X 0,Y 415.099,Z 897.897,A -85,B 0,C 180,E1 10068.622,E2 10068.622} C_VEL
LIN {X 0,Y 408.531,Z 918.566,A -85,B 0,C 180,E1 10068.011,E2 10068.011} C_VEL
LIN {X 0,Y 401.296,Z 938.441,A -85,B 0,C 180,E1 10067.309,E2 10067.309} C_VEL
LIN {X 0,Y 391.658,Z 961.798,A -85,B 0,C 180,E1 10066.317,E2 10066.317} C_VEL
LIN {X 0,Y 379.857,Z 986.547,A -85,B 0,C 180,E1 10065.019,E2 10065.019} C_VEL
LIN {X 0,Y 369.198,Z 1006.514,A -85,B 0,C 180,E1 10063.75,E2 10063.75} C_VEL
LIN {X 0,Y 358.735,Z 1024.427,A -85,B 0,C 180,E1 10062.404,E2 10062.404} C_VEL
LIN {X 0,Y 346.843,Z 1043.132,A -85,B 0,C 180,E1 10060.751,E2 10060.751} C_VEL
LIN {X 0,Y 330.951,Z 1065.871,A -85,B 0,C 180,E1 10058.279,E2 10058.279} C_VEL
LIN {X 0,Y 318.324,Z 1082.444,A -85,B 0,C 180,E1 10056.068,E2 10056.068} C_VEL
LIN {X 0,Y 306.552,Z 1096.983,A -85,B 0,C 180,E1 10053.759,E2 10053.759} C_VEL
LIN {X 0,Y 293.928,Z 1111.752,A -85,B 0,C 180,E1 10050.955,E2 10050.955} C_VEL
LIN {X 0,Y 278.478,Z 1128.876,A -85,B 0,C 180,E1 10046.923,E2 10046.923} C_VEL
LIN {X 0,Y 265.996,Z 1142.012,A -85,B 0,C 180,E1 10043.026,E2 10043.026} C_VEL
LIN {X 0,Y 255.411,Z 1152.938,A -85,B 0,C 180,E1 10039.072,E2 10039.072} C_VEL
LIN {X 0,Y 245.283,Z 1163.33,A -85,B 0,C 180,E1 10034.489,E2 10034.489} C_VEL
LIN {X 0,Y 234.18,Z 1174.958,A -85,B 0,C 180,E1 10027.939,E2 10027.939} C_VEL
LIN {X 0,Y 227.356,Z 1182.516,A -85,B 0,C 180,E1 10022.447,E2 10022.447} C_VEL
LIN {X 0,Y 222.453,Z 1188.538,A -85,B 0,C 180,E1 10016.998,E2 10016.998} C_VEL
LIN {X 0,Y 219.06,Z 1193.43,A -85,B 0,C 180,E1 10011.416,E2 10011.416} C_VEL
LIN {X 0,Y 216.979,Z 1197.391,A -85,B 0,C 180,E1 10005.502,E2 10005.502} C_VEL
LIN {X 0,Y 216.05,Z 1200.53,A -85,B 0,C 180,E1 9998.785,E2 9998.785} C_VEL
LIN {X 0,Y 215.917,Z 1201.961,A -85,B 0,C 180,E1 9992.92,E2 9992.92} C_VEL
LIN {X 0,Y 215.913,Z 1202.342,A -85,B 0,C 180,E1 9987.877,E2 9987.877} C_VEL
LIN {X 0,Y 216.006,Z 1201.722,A -85,B 0,C 180,E1 9982.141,E2 9982.141} C_VEL
LIN {X 0,Y 216.714,Z 1199.834,A -85,B 0,C 180,E1 9975.846,E2 9975.846} C_VEL
LIN {X 0,Y 218.556,Z 1196.963,A -85,B 0,C 180,E1 9969.933,E2 9969.933} C_VEL
LIN {X 0,Y 221.9,Z 1192.996,A -85,B 0,C 180,E1 9964.083,E2 9964.083} C_VEL
LIN {X 0,Y 226.9,Z 1187.907,A -85,B 0,C 180,E1 9958.373,E2 9958.373} C_VEL
LIN {X 0,Y 234.339,Z 1181.067,A -85,B 0,C 180,E1 9952.4,E2 9952.4} C_VEL
LIN {X 0,Y 245.611,Z 1171.198,A -85,B 0,C 180,E1 9945.883,E2 9945.883} C_VEL
LIN {X 0,Y 256.32,Z 1161.958,A -85,B 0,C 180,E1 9941.161,E2 9941.161} C_VEL
LIN {X 0,Y 267.358,Z 1152.376,A -85,B 0,C 180,E1 9937.196,E2 9937.196} C_VEL
LIN {X 0,Y 279.5,Z 1141.573,A -85,B 0,C 180,E1 9933.539,E2 9933.539} C_VEL
LIN {X 0,Y 294.797,Z 1127.484,A -85,B 0,C 180,E1 9929.683,E2 9929.683} C_VEL
LIN {X 0,Y 311.033,Z 1111.438,A -85,B 0,C 180,E1 9926.249,E2 9926.249} C_VEL
LIN {X 0,Y 324.542,Z 1097.291,A -85,B 0,C 180,E1 9923.794,E2 9923.794} C_VEL
LIN {X 0,Y 337.091,Z 1083.329,A -85,B 0,C 180,E1 9921.764,E2 9921.764} C_VEL
LIN {X 0,Y 350.152,Z 1067.816,A -85,B 0,C 180,E1 9919.866,E2 9919.866} C_VEL
LIN {X 0,Y 364.325,Z 1049.699,A -85,B 0,C 180,E1 9918.022,E2 9918.022} C_VEL
LIN {X 0,Y 380.45,Z 1026.903,A -85,B 0,C 180,E1 9916.144,E2 9916.144} C_VEL
LIN {X 0,Y 392.678,Z 1007.762,A -85,B 0,C 180,E1 9914.86,E2 9914.86} C_VEL
LIN {X 0,Y 403.136,Z 989.81,A -85,B 0,C 180,E1 9913.833,E2 9913.833} C_VEL
LIN {X 0,Y 412.926,Z 971.34,A -85,B 0,C 180,E1 9912.939,E2 9912.939} C_VEL
LIN {X 0,Y 422.366,Z 951.558,A -85,B 0,C 180,E1 9912.127,E2 9912.127} C_VEL
LIN {X 0,Y 432.814,Z 926.787,A -85,B 0,C 180,E1 9911.29,E2 9911.29} C_VEL
LIN {X 0,Y 441.732,Z 901.334,A -85,B 0,C 180,E1 9910.605,E2 9910.605} C_VEL
LIN {X 0,Y 448.166,Z 879.691,A -85,B 0,C 180,E1 9910.138,E2 9910.138} C_VEL
LIN {X 0,Y 453.561,Z 857.865,A -85,B 0,C 180,E1 9909.759,E2 9909.759} C_VEL
LIN {X 0,Y 458.842,Z 830.564,A -85,B 0,C 180,E1 9909.35,E2 9909.35} C_VEL
LIN {X 0,Y 464.244,Z 786.672,A -85,B 0,C 180,E1 9908.752,E2 9908.752} C_VEL
LIN {X 0,Y 480.023,Z 649.217,A -85,B 0,C 180,E1 9906.909,E2 9906.909} C_VEL
LIN {X 0,Y 479.255,Z 647.941,A -85,B 0,C 180,E1 9903.229,E2 9903.229} C_VEL
LIN {X 0,Y 479.988,Z 649.384,A -85,B 0,C 180,E1 9899.911,E2 9899.911} C_VEL
LIN {X 0,Y 460.021,Z 821.449,A -85,B 0,C 180,E1 9897.615,E2 9897.615} C_VEL
LIN {X 0,Y 455.638,Z 847.675,A -85,B 0,C 180,E1 9897.235,E2 9897.235} C_VEL
LIN {X 0,Y 449.214,Z 875.047,A -85,B 0,C 180,E1 9896.764,E2 9896.764} C_VEL
LIN {X 0,Y 443.109,Z 896.165,A -85,B 0,C 180,E1 9896.301,E2 9896.301} C_VEL
LIN {X 0,Y 436.132,Z 916.746,A -85,B 0,C 180,E1 9895.757,E2 9895.757} C_VEL
LIN {X 0,Y 428.481,Z 936.419,A -85,B 0,C 180,E1 9895.135,E2 9895.135} C_VEL
LIN {X 0,Y 418.993,Z 957.931,A -85,B 0,C 180,E1 9894.324,E2 9894.324} C_VEL
LIN {X 0,Y 405.857,Z 983.786,A -85,B 0,C 180,E1 9893.128,E2 9893.128} C_VEL
LIN {X 0,Y 394.752,Z 1003.114,A -85,B 0,C 180,E1 9892.035,E2 9892.035} C_VEL
LIN {X 0,Y 383.453,Z 1021.007,A -85,B 0,C 180,E1 9890.847,E2 9890.847} C_VEL
LIN {X 0,Y 371.152,Z 1038.867,A -85,B 0,C 180,E1 9889.444,E2 9889.444} C_VEL
LIN {X 0,Y 355.793,Z 1059.343,A -85,B 0,C 180,E1 9887.503,E2 9887.503} C_VEL
LIN {X 0,Y 339.73,Z 1078.536,A -85,B 0,C 180,E1 9885.23,E2 9885.23} C_VEL
LIN {X 0,Y 326.285,Z 1093.494,A -85,B 0,C 180,E1 9883.075,E2 9883.075} C_VEL
LIN {X 0,Y 313.453,Z 1106.893,A -85,B 0,C 180,E1 9880.766,E2 9880.766} C_VEL
LIN {X 0,Y 299.828,Z 1120.329,A -85,B 0,C 180,E1 9877.982,E2 9877.982} C_VEL
LIN {X 0,Y 282.856,Z 1136.111,A -85,B 0,C 180,E1 9873.877,E2 9873.877} C_VEL
LIN {X 0,Y 269.259,Z 1148.031,A -85,B 0,C 180,E1 9869.907,E2 9869.907} C_VEL
LIN {X 0,Y 257.548,Z 1158.015,A -85,B 0,C 180,E1 9865.783,E2 9865.783} C_VEL
LIN {X 0,Y 246.726,Z 1167.148,A -85,B 0,C 180,E1 9861.085,E2 9861.085} C_VEL
LIN {X 0,Y 235.168,Z 1176.971,A -85,B 0,C 180,E1 9854.55,E2 9854.55} C_VEL
LIN {X 0,Y 227.559,Z 1183.671,A -85,B 0,C 180,E1 9848.603,E2 9848.603} C_VEL
LIN {X 0,Y 222.423,Z 1188.606,A -85,B 0,C 180,E1 9842.952,E2 9842.952} C_VEL
LIN {X 0,Y 218.959,Z 1192.429,A -85,B 0,C 180,E1 9837.171,E2 9837.171} C_VEL
LIN {X 0,Y 216.987,Z 1195.142,A -85,B 0,C 180,E1 9831.435,E2 9831.435} C_VEL
LIN {X 0,Y 216.138,Z 1196.881,A -85,B 0,C 180,E1 9825.564,E2 9825.564} C_VEL
LIN {X 0,Y 215.931,Z 1197.566,A -85,B 0,C 180,E1 9819.865,E2 9819.865} C_VEL
LIN {X 0,Y 215.92,Z 1197.277,A -85,B 0,C 180,E1 9814.515,E2 9814.515} C_VEL
LIN {X 0,Y 216.083,Z 1195.966,A -85,B 0,C 180,E1 9808.674,E2 9808.674} C_VEL
LIN {X 0,Y 217.007,Z 1193.119,A -85,B 0,C 180,E1 9802.055,E2 9802.055} C_VEL
LIN {X 0,Y 219.26,Z 1189.04,A -85,B 0,C 180,E1 9795.745,E2 9795.745} C_VEL
LIN {X 0,Y 222.597,Z 1184.417,A -85,B 0,C 180,E1 9790.313,E2 9790.313} C_VEL
LIN {X 0,Y 227.609,Z 1178.454,A -85,B 0,C 180,E1 9784.779,E2 9784.779} C_VEL
LIN {X 0,Y 234.21,Z 1171.312,A -85,B 0,C 180,E1 9779.468,E2 9779.468} C_VEL
LIN {X 0,Y 244.058,Z 1161.311,A -85,B 0,C 180,E1 9773.556,E2 9773.556} C_VEL
LIN {X 0,Y 255.453,Z 1149.723,A -85,B 0,C 180,E1 9768.288,E2 9768.288} C_VEL
LIN {X 0,Y 265.847,Z 1139.161,A -85,B 0,C 180,E1 9764.39,E2 9764.39} C_VEL
LIN {X 0,Y 277.265,Z 1127.293,A -85,B 0,C 180,E1 9760.774,E2 9760.774} C_VEL
LIN {X 0,Y 291.542,Z 1111.936,A -85,B 0,C 180,E1 9756.958,E2 9756.958} C_VEL
LIN {X 0,Y 306.187,Z 1094.956,A -85,B 0,C 180,E1 9753.623,E2 9753.623} C_VEL
LIN {X 0,Y 318.368,Z 1080.052,A -85,B 0,C 180,E1 9751.213,E2 9751.213} C_VEL
LIN {X 0,Y 330.181,Z 1064.668,A -85,B 0,C 180,E1 9749.116,E2 9749.116} C_VEL
LIN {X 0,Y 344.616,Z 1044.513,A -85,B 0,C 180,E1 9746.828,E2 9746.828} C_VEL
LIN {X 0,Y 358.21,Z 1023.343,A -85,B 0,C 180,E1 9744.885,E2 9744.885} C_VEL
LIN {X 0,Y 368.973,Z 1005.046,A -85,B 0,C 180,E1 9743.476,E2 9743.476} C_VEL
LIN {X 0,Y 379.167,Z 986.11,A -85,B 0,C 180,E1 9742.244,E2 9742.244} C_VEL
LIN {X 0,Y 389.071,Z 965.754,A -85,B 0,C 180,E1 9741.116,E2 9741.116} C_VEL
LIN {X 0,Y 400.393,Z 939.232,A -85,B 0,C 180,E1 9739.917,E2 9739.917} C_VEL
LIN {X 0,Y 408.446,Z 917.278,A -85,B 0,C 180,E1 9739.107,E2 9739.107} C_VEL
LIN {X 0,Y 415.077,Z 896.478,A -85,B 0,C 180,E1 9738.472,E2 9738.472} C_VEL
LIN {X 0,Y 421.05,Z 874.481,A -85,B 0,C 180,E1 9737.918,E2 9737.918} C_VEL
LIN {X 0,Y 427.055,Z 847.164,A -85,B 0,C 180,E1 9737.377,E2 9737.377} C_VEL
LIN {X 0,Y 431.11,Z 821.035,A -85,B 0,C 180,E1 9736.959,E2 9736.959} C_VEL
LIN {X 0,Y 447.681,Z 662.24,A -85,B 0,C 180,E1 9734.704,E2 9734.704} C_VEL
LIN {X 0,Y 447.703,Z 662.025,A -85,B 0,C 180,E1 9734.701,E2 9734.701} C_VEL
LIN {X 0,Y 448.032,Z 657.033,A -85,B 0,C 180,E1 9734.504,E2 9734.504} C_VEL
LIN {X 0,Y 448.215,Z 644.656,A -85,B 0,C 180,E1 9733.545,E2 9733.545} C_VEL
LIN {X 0,Y 448.544,Z 640.346,A -85,B 0,C 180,E1 9733.389,E2 9733.389} C_VEL
LIN {X 0,Y 449.347,Z 632.43,A -85,B 0,C 180,E1 9733.25,E2 9733.25} C_VEL
LIN {X 0,Y 447.651,Z 628.995,A -85,B 0,C 180,E1 9731.467,E2 9731.467} C_VEL
LIN {X 0,Y 446.41,Z 626.271,A -85,B 0,C 180,E1 9729.801,E2 9729.801} C_VEL
LIN {X 0,Y 445.051,Z 622.891,A -85,B 0,C 180,E1 9727.098,E2 9727.098} C_VEL
LIN {X 0,Y 444.342,Z 622.087,A -85,B 0,C 180,E1 9722.967,E2 9722.967} C_VEL
LIN {X 0,Y 445.158,Z 623.076,A -85,B 0,C 180,E1 9719.743,E2 9719.743} C_VEL
LIN {X 0,Y 447.097,Z 627.674,A -85,B 0,C 180,E1 9716.346,E2 9716.346} C_VEL
LIN {X 0,Y 449.07,Z 631.873,A -85,B 0,C 180,E1 9714.121,E2 9714.121} C_VEL
LIN {X 0,Y 449.387,Z 632.82,A -85,B 0,C 180,E1 9713.787,E2 9713.787} C_VEL
LIN {X 0,Y 429.244,Z 822.711,A -85,B 0,C 180,E1 9711.129,E2 9711.129} C_VEL
LIN {X 0,Y 425.303,Z 847.986,A -85,B 0,C 180,E1 9710.732,E2 9710.732} C_VEL
LIN {X 0,Y 419.043,Z 876.33,A -85,B 0,C 180,E1 9710.209,E2 9710.209} C_VEL
LIN {X 0,Y 413.098,Z 897.948,A -85,B 0,C 180,E1 9709.7,E2 9709.7} C_VEL
LIN {X 0,Y 406.575,Z 918.224,A -85,B 0,C 180,E1 9709.117,E2 9709.117} C_VEL
LIN {X 0,Y 399.069,Z 938.571,A -85,B 0,C 180,E1 9708.418,E2 9708.418} C_VEL
LIN {X 0,Y 389.251,Z 962.009,A -85,B 0,C 180,E1 9707.446,E2 9707.446} C_VEL
LIN {X 0,Y 377.401,Z 986.457,A -85,B 0,C 180,E1 9706.193,E2 9706.193} C_VEL
LIN {X 0,Y 366.525,Z 1006.498,A -85,B 0,C 180,E1 9704.947,E2 9704.947} C_VEL
LIN {X 0,Y 355.874,Z 1024.402,A -85,B 0,C 180,E1 9703.631,E2 9703.631} C_VEL
LIN {X 0,Y 343.346,Z 1043.726,A -85,B 0,C 180,E1 9701.952,E2 9701.952} C_VEL
LIN {X 0,Y 327.533,Z 1065.833,A -85,B 0,C 180,E1 9699.582,E2 9699.582} C_VEL
LIN {X 0,Y 314.998,Z 1081.928,A -85,B 0,C 180,E1 9697.47,E2 9697.47} C_VEL
LIN {X 0,Y 302.176,Z 1097.371,A -85,B 0,C 180,E1 9695.043,E2 9695.043} C_VEL
LIN {X 0,Y 288.516,Z 1112.892,A -85,B 0,C 180,E1 9692.092,E2 9692.092} C_VEL
LIN {X 0,Y 272.41,Z 1130.049,A -85,B 0,C 180,E1 9687.98,E2 9687.98} C_VEL
LIN {X 0,Y 260.25,Z 1142.396,A -85,B 0,C 180,E1 9684.268,E2 9684.268} C_VEL
LIN {X 0,Y 249.413,Z 1153.146,A -85,B 0,C 180,E1 9680.326,E2 9680.326} C_VEL
LIN {X 0,Y 238.442,Z 1163.936,A -85,B 0,C 180,E1 9675.468,E2 9675.468} C_VEL
LIN {X 0,Y 227.236,Z 1175.075,A -85,B 0,C 180,E1 9668.992,E2 9668.992} C_VEL
LIN {X 0,Y 220.335,Z 1182.295,A -85,B 0,C 180,E1 9663.616,E2 9663.616} C_VEL
LIN {X 0,Y 215.074,Z 1188.339,A -85,B 0,C 180,E1 9658.004,E2 9658.004} C_VEL
LIN {X 0,Y 211.392,Z 1193.253,A -85,B 0,C 180,E1 9652.234,E2 9652.234} C_VEL
LIN {X 0,Y 209.188,Z 1197.072,A -85,B 0,C 180,E1 9646.38,E2 9646.38} C_VEL
LIN {X 0,Y 208.146,Z 1199.939,A -85,B 0,C 180,E1 9640.238,E2 9640.238} C_VEL
LIN {X 0,Y 207.922,Z 1201.597,A -85,B 0,C 180,E1 9634.413,E2 9634.413} C_VEL
LIN {X 0,Y 207.919,Z 1202.179,A -85,B 0,C 180,E1 9629.173,E2 9629.173} C_VEL
LIN {X 0,Y 207.952,Z 1201.906,A -85,B 0,C 180,E1 9623.651,E2 9623.651} C_VEL
LIN {X 0,Y 208.409,Z 1200.583,A -85,B 0,C 180,E1 9617.532,E2 9617.532} C_VEL
LIN {X 0,Y 210.394,Z 1197.548,A -85,B 0,C 180,E1 9610.219,E2 9610.219} C_VEL
LIN {X 0,Y 214.075,Z 1193.406,A -85,B 0,C 180,E1 9603.659,E2 9603.659} C_VEL
LIN {X 0,Y 219.281,Z 1188.434,A -85,B 0,C 180,E1 9597.759,E2 9597.759} C_VEL
LIN {X 0,Y 225.938,Z 1182.616,A -85,B 0,C 180,E1 9592.36,E2 9592.36} C_VEL
LIN {X 0,Y 234.663,Z 1175.359,A -85,B 0,C 180,E1 9587.021,E2 9587.021} C_VEL
LIN {X 0,Y 247.146,Z 1165.248,A -85,B 0,C 180,E1 9581.194,E2 9581.194} C_VEL
LIN {X 0,Y 261.18,Z 1153.533,A -85,B 0,C 180,E1 9576.123,E2 9576.123} C_VEL
LIN {X 0,Y 273.665,Z 1142.873,A -85,B 0,C 180,E1 9572.438,E2 9572.438} C_VEL
LIN {X 0,Y 287.135,Z 1130.907,A -85,B 0,C 180,E1 9569.07,E2 9569.07} C_VEL
LIN {X 0,Y 302.981,Z 1116.145,A -85,B 0,C 180,E1 9565.721,E2 9565.721} C_VEL
LIN {X 0,Y 320.515,Z 1098.417,A -85,B 0,C 180,E1 9562.575,E2 9562.575} C_VEL
LIN {X 0,Y 334.042,Z 1083.762,A -85,B 0,C 180,E1 9560.467,E2 9560.467} C_VEL
LIN {X 0,Y 347.154,Z 1068.553,A -85,B 0,C 180,E1 9558.636,E2 9558.636} C_VEL
LIN {X 0,Y 360.607,Z 1051.754,A -85,B 0,C 180,E1 9556.946,E2 9556.946} C_VEL
LIN {X 0,Y 376.108,Z 1030.708,A -85,B 0,C 180,E1 9555.202,E2 9555.202} C_VEL
LIN {X 0,Y 390.534,Z 1008.607,A -85,B 0,C 180,E1 9553.733,E2 9553.733} C_VEL
LIN {X 0,Y 401.292,Z 990.472,A -85,B 0,C 180,E1 9552.72,E2 9552.72} C_VEL
LIN {X 0,Y 411.209,Z 972.082,A -85,B 0,C 180,E1 9551.852,E2 9551.852} C_VEL
LIN {X 0,Y 420.763,Z 952.394,A -85,B 0,C 180,E1 9551.066,E2 9551.066} C_VEL
LIN {X 0,Y 430.867,Z 928.879,A -85,B 0,C 180,E1 9550.289,E2 9550.289} C_VEL
LIN {X 0,Y 440.346,Z 902.596,A -85,B 0,C 180,E1 9549.594,E2 9549.594} C_VEL
LIN {X 0,Y 447.048,Z 880.445,A -85,B 0,C 180,E1 9549.128,E2 9549.128} C_VEL
LIN {X 0,Y 452.478,Z 858.87,A -85,B 0,C 180,E1 9548.764,E2 9548.764} C_VEL
LIN {X 0,Y 457.276,Z 834.836,A -85,B 0,C 180,E1 9548.411,E2 9548.411} C_VEL
LIN {X 0,Y 462.154,Z 798.818,A -85,B 0,C 180,E1 9547.923,E2 9547.923} C_VEL
LIN {X 0,Y 478.704,Z 656.736,A -85,B 0,C 180,E1 9546.055,E2 9546.055} C_VEL
LIN {X 0,Y 478.285,Z 655.92,A -85,B 0,C 180,E1 9542.996,E2 9542.996} C_VEL
LIN {X 0,Y 478.675,Z 656.866,A -85,B 0,C 180,E1 9540.772,E2 9540.772} C_VEL
LIN {X 0,Y 459.237,Z 821.644,A -85,B 0,C 180,E1 9538.609,E2 9538.609} C_VEL
LIN {X 0,Y 454.68,Z 848.498,A -85,B 0,C 180,E1 9538.23,E2 9538.23} C_VEL
LIN {X 0,Y 448.21,Z 875.548,A -85,B 0,C 180,E1 9537.777,E2 9537.777} C_VEL
LIN {X 0,Y 441.919,Z 896.983,A -85,B 0,C 180,E1 9537.32,E2 9537.32} C_VEL
LIN {X 0,Y 434.892,Z 917.399,A -85,B 0,C 180,E1 9536.796,E2 9536.796} C_VEL
LIN {X 0,Y 426.625,Z 938.28,A -85,B 0,C 180,E1 9536.152,E2 9536.152} C_VEL
LIN {X 0,Y 415.383,Z 963.043,A -85,B 0,C 180,E1 9535.222,E2 9535.222} C_VEL
LIN {X 0,Y 403.318,Z 985.87,A -85,B 0,C 180,E1 9534.166,E2 9534.166} C_VEL
LIN {X 0,Y 392.282,Z 1004.665,A -85,B 0,C 180,E1 9533.119,E2 9533.119} C_VEL
LIN {X 0,Y 381.288,Z 1021.729,A -85,B 0,C 180,E1 9532.011,E2 9532.011} C_VEL
LIN {X 0,Y 368.442,Z 1040.009,A -85,B 0,C 180,E1 9530.602,E2 9530.602} C_VEL
LIN {X 0,Y 351.906,Z 1061.401,A -85,B 0,C 180,E1 9528.589,E2 9528.589} C_VEL
LIN {X 0,Y 336.592,Z 1079.271,A -85,B 0,C 180,E1 9526.494,E2 9526.494} C_VEL
LIN {X 0,Y 323.446,Z 1093.552,A -85,B 0,C 180,E1 9524.472,E2 9524.472} C_VEL
LIN {X 0,Y 309.899,Z 1107.34,A -85,B 0,C 180,E1 9522.135,E2 9522.135} C_VEL
LIN {X 0,Y 294.401,Z 1122.176,A -85,B 0,C 180,E1 9519.062,E2 9519.062} C_VEL
LIN {X 0,Y 277.014,Z 1137.634,A -85,B 0,C 180,E1 9514.953,E2 9514.953} C_VEL
LIN {X 0,Y 264.004,Z 1148.619,A -85,B 0,C 180,E1 9511.249,E2 9511.249} C_VEL
LIN {X 0,Y 252.142,Z 1158.307,A -85,B 0,C 180,E1 9507.212,E2 9507.212} C_VEL
LIN {X 0,Y 240.496,Z 1167.673,A -85,B 0,C 180,E1 9502.326,E2 9502.326} C_VEL
LIN {X 0,Y 228.038,Z 1177.648,A -85,B 0,C 180,E1 9495.447,E2 9495.447} C_VEL
LIN {X 0,Y 220.537,Z 1183.872,A -85,B 0,C 180,E1 9489.736,E2 9489.736} C_VEL
LIN {X 0,Y 215.026,Z 1188.784,A -85,B 0,C 180,E1 9483.917,E2 9483.917} C_VEL
LIN {X 0,Y 211.27,Z 1192.587,A -85,B 0,C 180,E1 9477.939,E2 9477.939} C_VEL
LIN {X 0,Y 209.087,Z 1195.316,A -85,B 0,C 180,E1 9471.901,E2 9471.901} C_VEL
LIN {X 0,Y 208.119,Z 1197.134,A -85,B 0,C 180,E1 9465.321,E2 9465.321} C_VEL
LIN {X 0,Y 207.929,Z 1197.708,A -85,B 0,C 180,E1 9459.41,E2 9459.41} C_VEL
LIN {X 0,Y 207.922,Z 1197.31,A -85,B 0,C 180,E1 9453.86,E2 9453.86} C_VEL
LIN {X 0,Y 208.145,Z 1195.866,A -85,B 0,C 180,E1 9447.798,E2 9447.798} C_VEL
LIN {X 0,Y 209.281,Z 1192.826,A -85,B 0,C 180,E1 9440.929,E2 9440.929} C_VEL
LIN {X 0,Y 211.601,Z 1189.042,A -85,B 0,C 180,E1 9434.937,E2 9434.937} C_VEL
LIN {X 0,Y 215.217,Z 1184.4,A -85,B 0,C 180,E1 9429.324,E2 9429.324} C_VEL
LIN {X 0,Y 220.308,Z 1178.714,A -85,B 0,C 180,E1 9423.882,E2 9423.882} C_VEL
LIN {X 0,Y 226.904,Z 1171.944,A -85,B 0,C 180,E1 9418.67,E2 9418.67} C_VEL
LIN {X 0,Y 236.033,Z 1163.074,A -85,B 0,C 180,E1 9413.193,E2 9413.193} C_VEL
LIN {X 0,Y 248.535,Z 1150.996,A -85,B 0,C 180,E1 9407.412,E2 9407.412} C_VEL
LIN {X 0,Y 259.911,Z 1139.88,A -85,B 0,C 180,E1 9403.218,E2 9403.218} C_VEL
LIN {X 0,Y 271.42,Z 1128.349,A -85,B 0,C 180,E1 9399.654,E2 9399.654} C_VEL
LIN {X 0,Y 284.099,Z 1115.158,A -85,B 0,C 180,E1 9396.299,E2 9396.299} C_VEL
LIN {X 0,Y 300.424,Z 1097.108,A -85,B 0,C 180,E1 9392.628,E2 9392.628} C_VEL
LIN {X 0,Y 313.295,Z 1081.833,A -85,B 0,C 180,E1 9390.132,E2 9390.132} C_VEL
LIN {X 0,Y 325.29,Z 1066.672,A -85,B 0,C 180,E1 9388.054,E2 9388.054} C_VEL
LIN {X 0,Y 337.089,Z 1050.694,A -85,B 0,C 180,E1 9386.2,E2 9386.2} C_VEL
LIN {X 0,Y 349.632,Z 1032.381,A -85,B 0,C 180,E1 9384.415,E2 9384.415} C_VEL
LIN {X 0,Y 364.657,Z 1008.03,A -85,B 0,C 180,E1 9382.479,E2 9382.479} C_VEL
LIN {X 0,Y 375.398,Z 988.629,A -85,B 0,C 180,E1 9381.218,E2 9381.218} C_VEL
LIN {X 0,Y 384.595,Z 970.299,A -85,B 0,C 180,E1 9380.197,E2 9380.197} C_VEL
LIN {X 0,Y 393.494,Z 950.661,A -85,B 0,C 180,E1 9379.271,E2 9379.271} C_VEL
LIN {X 0,Y 403.358,Z 926.095,A -85,B 0,C 180,E1 9378.307,E2 9378.307} C_VEL
LIN {X 0,Y 411.996,Z 900.242,A -85,B 0,C 180,E1 9377.493,E2 9377.493} C_VEL
LIN {X 0,Y 418.159,Z 878.416,A -85,B 0,C 180,E1 9376.94,E2 9376.94} C_VEL
LIN {X 0,Y 423.183,Z 857.055,A -85,B 0,C 180,E1 9376.501,E2 9376.501} C_VEL
LIN {X 0,Y 427.759,Z 832.48,A -85,B 0,C 180,E1 9376.09,E2 9376.09} C_VEL
LIN {X 0,Y 432.184,Z 796.189,A -85,B 0,C 180,E1 9375.558,E2 9375.558} C_VEL
LIN {X 0,Y 448.544,Z 640.346,A -85,B 0,C 180,E1 9373.389,E2 9373.389} C_VEL
LIN {X 0,Y 448.618,Z 638.14,A -85,B 0,C 180,E1 9373.238,E2 9373.238} C_VEL
LIN {X 0,Y 448.363,Z 636.402,A -85,B 0,C 180,E1 9372.871,E2 9372.871} C_VEL
LIN {X 0,Y 447.699,Z 635.508,A -85,B 0,C 180,E1 9372.234,E2 9372.234} C_VEL
LIN {X 0,Y 446.096,Z 635.63,A -85,B 0,C 180,E1 9370.745,E2 9370.745} C_VEL
LIN {X 0,Y 445.833,Z 635.188,A -85,B 0,C 180,E1 9370.406,E2 9370.406} C_VEL
LIN {X 0,Y 444.023,Z 630.801,A -85,B 0,C 180,E1 9366.985,E2 9366.985} C_VEL
LIN {X 0,Y 443.364,Z 630.028,A -85,B 0,C 180,E1 9362.973,E2 9362.973} C_VEL
LIN {X 0,Y 444.162,Z 631.149,A -85,B 0,C 180,E1 9359.742,E2 9359.742} C_VEL
LIN {X 0,Y 445.956,Z 635.468,A -85,B 0,C 180,E1 9356.529,E2 9356.529} C_VEL
LIN {X 0,Y 447.461,Z 638.875,A -85,B 0,C 180,E1 9354.717,E2 9354.717} C_VEL
LIN {X 0,Y 427.604,Z 822.765,A -85,B 0,C 180,E1 9352.179,E2 9352.179} C_VEL
LIN {X 0,Y 423.507,Z 848.615,A -85,B 0,C 180,E1 9351.781,E2 9351.781} C_VEL
LIN {X 0,Y 417.232,Z 876.509,A -85,B 0,C 180,E1 9351.279,E2 9351.279} C_VEL
LIN {X 0,Y 411.245,Z 897.996,A -85,B 0,C 180,E1 9350.787,E2 9350.787} C_VEL
LIN {X 0,Y 404.554,Z 918.505,A -85,B 0,C 180,E1 9350.213,E2 9350.213} C_VEL
LIN {X 0,Y 396.896,Z 938.946,A -85,B 0,C 180,E1 9349.529,E2 9349.529} C_VEL
LIN {X 0,Y 386.636,Z 963.038,A -85,B 0,C 180,E1 9348.552,E2 9348.552} C_VEL
LIN {X 0,Y 374.617,Z 987.271,A -85,B 0,C 180,E1 9347.331,E2 9347.331} C_VEL
LIN {X 0,Y 364.184,Z 1006.187,A -85,B 0,C 180,E1 9346.18,E2 9346.18} C_VEL
LIN {X 0,Y 353.179,Z 1024.377,A -85,B 0,C 180,E1 9344.878,E2 9344.878} C_VEL
LIN {X 0,Y 340.421,Z 1043.693,A -85,B 0,C 180,E1 9343.235,E2 9343.235} C_VEL
LIN {X 0,Y 324.423,Z 1065.617,A -85,B 0,C 180,E1 9340.931,E2 9340.931} C_VEL
LIN {X 0,Y 311.079,Z 1082.361,A -85,B 0,C 180,E1 9338.765,E2 9338.765} C_VEL
LIN {X 0,Y 298.714,Z 1096.892,A -85,B 0,C 180,E1 9336.51,E2 9336.51} C_VEL
LIN {X 0,Y 285.381,Z 1111.656,A -85,B 0,C 180,E1 9333.756,E2 9333.756} C_VEL
LIN {X 0,Y 269.349,Z 1128.366,A -85,B 0,C 180,E1 9329.874,E2 9329.874} C_VEL
LIN {X 0,Y 255.828,Z 1141.628,A -85,B 0,C 180,E1 9325.951,E2 9325.951} C_VEL
LIN {X 0,Y 244.091,Z 1152.822,A -85,B 0,C 180,E1 9321.857,E2 9321.857} C_VEL
LIN {X 0,Y 233.091,Z 1163.171,A -85,B 0,C 180,E1 9317.181,E2 9317.181} C_VEL
LIN {X 0,Y 220.762,Z 1174.829,A -85,B 0,C 180,E1 9310.365,E2 9310.365} C_VEL
LIN {X 0,Y 213.102,Z 1182.383,A -85,B 0,C 180,E1 9304.591,E2 9304.591} C_VEL
LIN {X 0,Y 207.531,Z 1188.401,A -85,B 0,C 180,E1 9298.802,E2 9298.802} C_VEL
LIN {X 0,Y 203.762,Z 1193.076,A -85,B 0,C 180,E1 9293.114,E2 9293.114} C_VEL
LIN {X 0,Y 201.345,Z 1196.916,A -85,B 0,C 180,E1 9287.037,E2 9287.037} C_VEL
LIN {X 0,Y 200.18,Z 1199.804,A -85,B 0,C 180,E1 9280.65,E2 9280.65} C_VEL
LIN {X 0,Y 199.927,Z 1201.412,A -85,B 0,C 180,E1 9274.877,E2 9274.877} C_VEL
LIN {X 0,Y 199.923,Z 1202.06,A -85,B 0,C 180,E1 9269.427,E2 9269.427} C_VEL
LIN {X 0,Y 199.937,Z 1201.899,A -85,B 0,C 180,E1 9264.26,E2 9264.26} C_VEL
LIN {X 0,Y 200.222,Z 1201.011,A -85,B 0,C 180,E1 9259.061,E2 9259.061} C_VEL
LIN {X 0,Y 201.321,Z 1199.173,A -85,B 0,C 180,E1 9253.258,E2 9253.258} C_VEL
LIN {X 0,Y 203.752,Z 1196.273,A -85,B 0,C 180,E1 9247.19,E2 9247.19} C_VEL
LIN {X 0,Y 207.916,Z 1192.25,A -85,B 0,C 180,E1 9241.076,E2 9241.076} C_VEL
LIN {X 0,Y 214.778,Z 1186.42,A -85,B 0,C 180,E1 9234.415,E2 9234.415} C_VEL
LIN {X 0,Y 225.464,Z 1177.881,A -85,B 0,C 180,E1 9227.273,E2 9227.273} C_VEL
LIN {X 0,Y 236.23,Z 1169.504,A -85,B 0,C 180,E1 9221.972,E2 9221.972} C_VEL
LIN {X 0,Y 247.336,Z 1160.822,A -85,B 0,C 180,E1 9217.596,E2 9217.596} C_VEL
LIN {X 0,Y 260.091,Z 1150.62,A -85,B 0,C 180,E1 9213.467,E2 9213.467} C_VEL
LIN {X 0,Y 276.805,Z 1136.747,A -85,B 0,C 180,E1 9209.057,E2 9209.057} C_VEL
LIN {X 0,Y 292.677,Z 1122.592,A -85,B 0,C 180,E1 9205.593,E2 9205.593} C_VEL
LIN {X 0,Y 307.155,Z 1108.925,A -85,B 0,C 180,E1 9202.894,E2 9202.894} C_VEL
LIN {X 0,Y 321.448,Z 1094.557,A -85,B 0,C 180,E1 9200.568,E2 9200.568} C_VEL
LIN {X 0,Y 338.741,Z 1075.894,A -85,B 0,C 180,E1 9198.114,E2 9198.114} C_VEL
LIN {X 0,Y 355.3,Z 1056,A -85,B 0,C 180,E1 9196.05,E2 9196.05} C_VEL
LIN {X 0,Y 368.299,Z 1039.042,A -85,B 0,C 180,E1 9194.605,E2 9194.605} C_VEL
LIN {X 0,Y 380.263,Z 1022.068,A -85,B 0,C 180,E1 9193.377,E2 9193.377} C_VEL
LIN {X 0,Y 392.827,Z 1002.581,A -85,B 0,C 180,E1 9192.197,E2 9192.197} C_VEL
LIN {X 0,Y 407.354,Z 977.237,A -85,B 0,C 180,E1 9190.947,E2 9190.947} C_VEL
LIN {X 0,Y 417.921,Z 956.187,A -85,B 0,C 180,E1 9190.104,E2 9190.104} C_VEL
LIN {X 0,Y 426.773,Z 936.361,A -85,B 0,C 180,E1 9189.439,E2 9189.439} C_VEL
LIN {X 0,Y 434.945,Z 915.583,A -85,B 0,C 180,E1 9188.86,E2 9188.86} C_VEL
LIN {X 0,Y 443.092,Z 891.547,A -85,B 0,C 180,E1 9188.313,E2 9188.313} C_VEL
LIN {X 0,Y 450.66,Z 863.699,A -85,B 0,C 180,E1 9187.822,E2 9187.822} C_VEL
LIN {X 0,Y 455.539,Z 840.731,A -85,B 0,C 180,E1 9187.489,E2 9187.489} C_VEL
LIN {X 0,Y 459.146,Z 818.236,A -85,B 0,C 180,E1 9187.182,E2 9187.182} C_VEL
LIN {X 0,Y 477.485,Z 664.314,A -85,B 0,C 180,E1 9185.196,E2 9185.196} C_VEL
LIN {X 0,Y 477.344,Z 663.949,A -85,B 0,C 180,E1 9182.521,E2 9182.521} C_VEL
LIN {X 0,Y 477.455,Z 664.478,A -85,B 0,C 180,E1 9181.637,E2 9181.637} C_VEL
LIN {X 0,Y 458.619,Z 821.737,A -85,B 0,C 180,E1 9179.609,E2 9179.609} C_VEL
LIN {X 0,Y 454.025,Z 848.495,A -85,B 0,C 180,E1 9179.24,E2 9179.24} C_VEL
LIN {X 0,Y 447.47,Z 875.633,A -85,B 0,C 180,E1 9178.801,E2 9178.801} C_VEL
LIN {X 0,Y 441.116,Z 897.049,A -85,B 0,C 180,E1 9178.362,E2 9178.362} C_VEL
LIN {X 0,Y 433.991,Z 917.523,A -85,B 0,C 180,E1 9177.854,E2 9177.854} C_VEL
LIN {X 0,Y 425.44,Z 938.863,A -85,B 0,C 180,E1 9177.218,E2 9177.218} C_VEL
LIN {X 0,Y 413.803,Z 964.03,A -85,B 0,C 180,E1 9176.299,E2 9176.299} C_VEL
LIN {X 0,Y 402.275,Z 985.577,A -85,B 0,C 180,E1 9175.334,E2 9175.334} C_VEL
LIN {X 0,Y 390.874,Z 1004.748,A -85,B 0,C 180,E1 9174.303,E2 9174.303} C_VEL
LIN {X 0,Y 379.288,Z 1022.447,A -85,B 0,C 180,E1 9173.187,E2 9173.187} C_VEL
LIN {X 0,Y 365.189,Z 1042.115,A -85,B 0,C 180,E1 9171.699,E2 9171.699} C_VEL
LIN {X 0,Y 348.071,Z 1063.535,A -85,B 0,C 180,E1 9169.69,E2 9169.69} C_VEL
LIN {X 0,Y 333.96,Z 1079.641,A -85,B 0,C 180,E1 9167.828,E2 9167.828} C_VEL
LIN {X 0,Y 320.133,Z 1094.304,A -85,B 0,C 180,E1 9165.789,E2 9165.789} C_VEL
LIN {X 0,Y 305.714,Z 1108.577,A -85,B 0,C 180,E1 9163.39,E2 9163.39} C_VEL
LIN {X 0,Y 288.312,Z 1124.675,A -85,B 0,C 180,E1 9160.021,E2 9160.021} C_VEL
LIN {X 0,Y 271.989,Z 1138.57,A -85,B 0,C 180,E1 9156.255,E2 9156.255} C_VEL
LIN {X 0,Y 258.869,Z 1149.234,A -85,B 0,C 180,E1 9152.636,E2 9152.636} C_VEL
LIN {X 0,Y 246.299,Z 1159.071,A -85,B 0,C 180,E1 9148.484,E2 9148.484} C_VEL
LIN {X 0,Y 232.459,Z 1169.72,A -85,B 0,C 180,E1 9142.724,E2 9142.724} C_VEL
LIN {X 0,Y 220.948,Z 1178.341,A -85,B 0,C 180,E1 9136.39,E2 9136.39} C_VEL
LIN {X 0,Y 213.124,Z 1184.454,A -85,B 0,C 180,E1 9130.532,E2 9130.532} C_VEL
LIN {X 0,Y 207.225,Z 1189.382,A -85,B 0,C 180,E1 9124.369,E2 9124.369} C_VEL
LIN {X 0,Y 202.66,Z 1193.862,A -85,B 0,C 180,E1 9116.677,E2 9116.677} C_VEL
LIN {X 0,Y 200.539,Z 1196.446,A -85,B 0,C 180,E1 9109.212,E2 9109.212} C_VEL
LIN {X 0,Y 200.002,Z 1197.523,A -85,B 0,C 180,E1 9103.295,E2 9103.295} C_VEL
LIN {X 0,Y 199.914,Z 1197.71,A -85,B 0,C 180,E1 9097.761,E2 9097.761} C_VEL
LIN {X 0,Y 199.94,Z 1197.092,A -85,B 0,C 180,E1 9092.293,E2 9092.293} C_VEL
LIN {X 0,Y 200.282,Z 1195.457,A -85,B 0,C 180,E1 9086.279,E2 9086.279} C_VEL
LIN {X 0,Y 201.527,Z 1192.69,A -85,B 0,C 180,E1 9080,E2 9080} C_VEL
LIN {X 0,Y 203.981,Z 1189.044,A -85,B 0,C 180,E1 9074.068,E2 9074.068} C_VEL
LIN {X 0,Y 207.904,Z 1184.382,A -85,B 0,C 180,E1 9068.265,E2 9068.265} C_VEL
LIN {X 0,Y 213.361,Z 1178.675,A -85,B 0,C 180,E1 9062.661,E2 9062.661} C_VEL
LIN {X 0,Y 220.76,Z 1171.539,A -85,B 0,C 180,E1 9057.078,E2 9057.078} C_VEL
LIN {X 0,Y 231.632,Z 1161.552,A -85,B 0,C 180,E1 9050.934,E2 9050.934} C_VEL
LIN {X 0,Y 244.096,Z 1149.966,A -85,B 0,C 180,E1 9045.538,E2 9045.538} C_VEL
LIN {X 0,Y 255.328,Z 1139.409,A -85,B 0,C 180,E1 9041.587,E2 9041.587} C_VEL
LIN {X 0,Y 266.944,Z 1128.166,A -85,B 0,C 180,E1 9038.134,E2 9038.134} C_VEL
LIN {X 0,Y 280.73,Z 1114.256,A -85,B 0,C 180,E1 9034.641,E2 9034.641} C_VEL
LIN {X 0,Y 296.819,Z 1096.868,A -85,B 0,C 180,E1 9031.172,E2 9031.172} C_VEL
LIN {X 0,Y 310.071,Z 1081.513,A -85,B 0,C 180,E1 9028.707,E2 9028.707} C_VEL
LIN {X 0,Y 322.272,Z 1066.417,A -85,B 0,C 180,E1 9026.68,E2 9026.68} C_VEL
LIN {X 0,Y 334.582,Z 1050.059,A -85,B 0,C 180,E1 9024.828,E2 9024.828} C_VEL
LIN {X 0,Y 349.331,Z 1028.824,A -85,B 0,C 180,E1 9022.835,E2 9022.835} C_VEL
LIN {X 0,Y 362.514,Z 1007.446,A -85,B 0,C 180,E1 9021.213,E2 9021.213} C_VEL
LIN {X 0,Y 373.434,Z 987.967,A -85,B 0,C 180,E1 9019.984,E2 9019.984} C_VEL
LIN {X 0,Y 382.781,Z 969.547,A -85,B 0,C 180,E1 9018.991,E2 9018.991} C_VEL
LIN {X 0,Y 392.25,Z 948.824,A -85,B 0,C 180,E1 9018.05,E2 9018.05} C_VEL
LIN {X 0,Y 402.926,Z 921.889,A -85,B 0,C 180,E1 9017.049,E2 9017.049} C_VEL
LIN {X 0,Y 410.577,Z 898.939,A -85,B 0,C 180,E1 9016.365,E2 9016.365} C_VEL
LIN {X 0,Y 416.633,Z 877.584,A -85,B 0,C 180,E1 9015.844,E2 9015.844} C_VEL
LIN {X 0,Y 421.768,Z 855.8,A -85,B 0,C 180,E1 9015.414,E2 9015.414} C_VEL
LIN {X 0,Y 426.83,Z 828.125,A -85,B 0,C 180,E1 9014.969,E2 9014.969} C_VEL
LIN {X 0,Y 432.025,Z 782.761,A -85,B 0,C 180,E1 9014.327,E2 9014.327} C_VEL
LIN {X 0,Y 447.422,Z 638.58,A -85,B 0,C 180,E1 9012.323,E2 9012.323} C_VEL
LIN {X 0,Y 445.833,Z 635.188,A -85,B 0,C 180,E1 9010.406,E2 9010.406} C_VEL
LIN {X 0,Y 445.139,Z 634.508,A -85,B 0,C 180,E1 9009.49,E2 9009.49} C_VEL
LIN {X 0,Y 444.013,Z 635.908,A -85,B 0,C 180,E1 9008.141,E2 9008.141} C_VEL
LIN {X 0,Y 442.834,Z 638.289,A -85,B 0,C 180,E1 9006.341,E2 9006.341} C_VEL
LIN {X 0,Y 442.654,Z 638.352,A -85,B 0,C 180,E1 9005.83,E2 9005.83} C_VEL
LIN {X 0,Y 442.444,Z 638.101,A -85,B 0,C 180,E1 9002.331,E2 9002.331} C_VEL
LIN {X 0,Y 443.126,Z 639.03,A -85,B 0,C 180,E1 8999.871,E2 8999.871} C_VEL
LIN {X 0,Y 444.819,Z 643.26,A -85,B 0,C 180,E1 8996.714,E2 8996.714} C_VEL
LIN {X 0,Y 445.609,Z 645.33,A -85,B 0,C 180,E1 8995.65,E2 8995.65} C_VEL
LIN {X 0,Y 426.125,Z 822.684,A -85,B 0,C 180,E1 8993.239,E2 8993.239} C_VEL
LIN {X 0,Y 421.971,Z 848.549,A -85,B 0,C 180,E1 8992.849,E2 8992.849} C_VEL
LIN {X 0,Y 415.627,Z 876.435,A -85,B 0,C 180,E1 8992.363,E2 8992.363} C_VEL
LIN {X 0,Y 409.541,Z 898.017,A -85,B 0,C 180,E1 8991.885,E2 8991.885} C_VEL
LIN {X 0,Y 402.991,Z 917.893,A -85,B 0,C 180,E1 8991.347,E2 8991.347} C_VEL
LIN {X 0,Y 395.162,Z 938.593,A -85,B 0,C 180,E1 8990.678,E2 8990.678} C_VEL
LIN {X 0,Y 384.668,Z 962.934,A -85,B 0,C 180,E1 8989.722,E2 8989.722} C_VEL
LIN {X 0,Y 372.388,Z 987.335,A -85,B 0,C 180,E1 8988.526,E2 8988.526} C_VEL
LIN {X 0,Y 361.565,Z 1006.629,A -85,B 0,C 180,E1 8987.381,E2 8987.381} C_VEL
LIN {X 0,Y 350.622,Z 1024.394,A -85,B 0,C 180,E1 8986.14,E2 8986.14} C_VEL
LIN {X 0,Y 337.245,Z 1044.284,A -85,B 0,C 180,E1 8984.483,E2 8984.483} C_VEL
LIN {X 0,Y 320.932,Z 1066.11,A -85,B 0,C 180,E1 8982.222,E2 8982.222} C_VEL
LIN {X 0,Y 307.731,Z 1082.307,A -85,B 0,C 180,E1 8980.159,E2 8980.159} C_VEL
LIN {X 0,Y 294.676,Z 1097.276,A -85,B 0,C 180,E1 8977.866,E2 8977.866} C_VEL
LIN {X 0,Y 280.263,Z 1112.791,A -85,B 0,C 180,E1 8974.98,E2 8974.98} C_VEL
LIN {X 0,Y 263.129,Z 1129.937,A -85,B 0,C 180,E1 8970.923,E2 8970.923} C_VEL
LIN {X 0,Y 250.544,Z 1141.863,A -85,B 0,C 180,E1 8967.356,E2 8967.356} C_VEL
LIN {X 0,Y 238.951,Z 1152.497,A -85,B 0,C 180,E1 8963.455,E2 8963.455} C_VEL
LIN {X 0,Y 227.418,Z 1162.884,A -85,B 0,C 180,E1 8958.738,E2 8958.738} C_VEL
LIN {X 0,Y 214.827,Z 1174.218,A -85,B 0,C 180,E1 8952.083,E2 8952.083} C_VEL
LIN {X 0,Y 206.257,Z 1182.159,A -85,B 0,C 180,E1 8945.913,E2 8945.913} C_VEL
LIN {X 0,Y 200.508,Z 1187.938,A -85,B 0,C 180,E1 8940.241,E2 8940.241} C_VEL
LIN {X 0,Y 196.291,Z 1192.769,A -85,B 0,C 180,E1 8934.243,E2 8934.243} C_VEL
LIN {X 0,Y 193.617,Z 1196.596,A -85,B 0,C 180,E1 8928.05,E2 8928.05} C_VEL
LIN {X 0,Y 192.318,Z 1199.32,A -85,B 0,C 180,E1 8922.003,E2 8922.003} C_VEL
LIN {X 0,Y 191.96,Z 1200.952,A -85,B 0,C 180,E1 8916.58,E2 8916.58} C_VEL
LIN {X 0,Y 191.92,Z 1201.807,A -85,B 0,C 180,E1 8911.493,E2 8911.493} C_VEL
LIN {X 0,Y 191.916,Z 1201.988,A -85,B 0,C 180,E1 8906.116,E2 8906.116} C_VEL
LIN {X 0,Y 192.122,Z 1201.299,A -85,B 0,C 180,E1 8900.111,E2 8900.111} C_VEL
LIN {X 0,Y 193.238,Z 1199.477,A -85,B 0,C 180,E1 8893.466,E2 8893.466} C_VEL
LIN {X 0,Y 195.845,Z 1196.573,A -85,B 0,C 180,E1 8886.852,E2 8886.852} C_VEL
LIN {X 0,Y 200.049,Z 1192.78,A -85,B 0,C 180,E1 8880.672,E2 8880.672} C_VEL
LIN {X 0,Y 206.212,Z 1187.807,A -85,B 0,C 180,E1 8874.549,E2 8874.549} C_VEL
LIN {X 0,Y 214.572,Z 1181.492,A -85,B 0,C 180,E1 8868.571,E2 8868.571} C_VEL
LIN {X 0,Y 227.191,Z 1172.266,A -85,B 0,C 180,E1 8861.947,E2 8861.947} C_VEL
LIN {X 0,Y 241.114,Z 1161.846,A -85,B 0,C 180,E1 8856.44,E2 8856.44} C_VEL
LIN {X 0,Y 254.255,Z 1151.78,A -85,B 0,C 180,E1 8852.276,E2 8852.276} C_VEL
LIN {X 0,Y 268.568,Z 1140.382,A -85,B 0,C 180,E1 8848.525,E2 8848.525} C_VEL
LIN {X 0,Y 287.366,Z 1124.471,A -85,B 0,C 180,E1 8844.46,E2 8844.46} C_VEL
LIN {X 0,Y 303.233,Z 1109.951,A -85,B 0,C 180,E1 8841.59,E2 8841.59} C_VEL
LIN {X 0,Y 317.951,Z 1095.556,A -85,B 0,C 180,E1 8839.281,E2 8839.281} C_VEL
LIN {X 0,Y 332.876,Z 1079.885,A -85,B 0,C 180,E1 8837.22,E2 8837.22} C_VEL
LIN {X 0,Y 350.518,Z 1059.703,A -85,B 0,C 180,E1 8835.078,E2 8835.078} C_VEL
LIN {X 0,Y 365.734,Z 1040.331,A -85,B 0,C 180,E1 8833.438,E2 8833.438} C_VEL
LIN {X 0,Y 378.215,Z 1022.977,A -85,B 0,C 180,E1 8832.21,E2 8832.21} C_VEL
LIN {X 0,Y 390.277,Z 1004.641,A -85,B 0,C 180,E1 8831.124,E2 8831.124} C_VEL
LIN {X 0,Y 403.136,Z 983.037,A -85,B 0,C 180,E1 8830.057,E2 8830.057} C_VEL
LIN {X 0,Y 416.131,Z 958.01,A -85,B 0,C 180,E1 8829.059,E2 8829.059} C_VEL
LIN {X 0,Y 425.693,Z 936.973,A -85,B 0,C 180,E1 8828.374,E2 8828.374} C_VEL
LIN {X 0,Y 434.016,Z 916.119,A -85,B 0,C 180,E1 8827.812,E2 8827.812} C_VEL
LIN {X 0,Y 442.019,Z 892.854,A -85,B 0,C 180,E1 8827.299,E2 8827.299} C_VEL
LIN {X 0,Y 449.984,Z 864.165,A -85,B 0,C 180,E1 8826.809,E2 8826.809} C_VEL
LIN {X 0,Y 454.969,Z 841.014,A -85,B 0,C 180,E1 8826.484,E2 8826.484} C_VEL
LIN {X 0,Y 458.62,Z 818.633,A -85,B 0,C 180,E1 8826.186,E2 8826.186} C_VEL
LIN {X 0,Y 476.366,Z 671.918,A -85,B 0,C 180,E1 8824.303,E2 8824.303} C_VEL
LIN {X 0,Y 476.347,Z 672.058,A -85,B 0,C 180,E1 8822.508,E2 8822.508} C_VEL
LIN {X 0,Y 458.128,Z 821.91,A -85,B 0,C 180,E1 8820.609,E2 8820.609} C_VEL
LIN {X 0,Y 453.412,Z 849.027,A -85,B 0,C 180,E1 8820.245,E2 8820.245} C_VEL
LIN {X 0,Y 446.812,Z 875.965,A -85,B 0,C 180,E1 8819.825,E2 8819.825} C_VEL
LIN {X 0,Y 440.46,Z 897.152,A -85,B 0,C 180,E1 8819.407,E2 8819.407} C_VEL
LIN {X 0,Y 433.317,Z 917.473,A -85,B 0,C 180,E1 8818.922,E2 8818.922} C_VEL
LIN {X 0,Y 425.116,Z 937.773,A -85,B 0,C 180,E1 8818.342,E2 8818.342} C_VEL
LIN {X 0,Y 413.836,Z 962.229,A -85,B 0,C 180,E1 8817.495,E2 8817.495} C_VEL
LIN {X 0,Y 401.194,Z 985.64,A -85,B 0,C 180,E1 8816.491,E2 8816.491} C_VEL
LIN {X 0,Y 390.125,Z 1004.055,A -85,B 0,C 180,E1 8815.539,E2 8815.539} C_VEL
LIN {X 0,Y 378.219,Z 1022.048,A -85,B 0,C 180,E1 8814.449,E2 8814.449} C_VEL
LIN {X 0,Y 364.961,Z 1040.339,A -85,B 0,C 180,E1 8813.121,E2 8813.121} C_VEL
LIN {X 0,Y 347.552,Z 1062.041,A -85,B 0,C 180,E1 8811.188,E2 8811.188} C_VEL
LIN {X 0,Y 332.697,Z 1078.748,A -85,B 0,C 180,E1 8809.338,E2 8809.338} C_VEL
LIN {X 0,Y 318.651,Z 1093.389,A -85,B 0,C 180,E1 8807.382,E2 8807.382} C_VEL
LIN {X 0,Y 304.175,Z 1107.448,A -85,B 0,C 180,E1 8805.107,E2 8805.107} C_VEL
LIN {X 0,Y 288.22,Z 1121.924,A -85,B 0,C 180,E1 8802.224,E2 8802.224} C_VEL
LIN {X 0,Y 269.748,Z 1137.417,A -85,B 0,C 180,E1 8798.243,E2 8798.243} C_VEL
LIN {X 0,Y 255.277,Z 1148.785,A -85,B 0,C 180,E1 8794.478,E2 8794.478} C_VEL
LIN {X 0,Y 242.466,Z 1158.431,A -85,B 0,C 180,E1 8790.47,E2 8790.47} C_VEL
LIN {X 0,Y 229.982,Z 1167.543,A -85,B 0,C 180,E1 8785.693,E2 8785.693} C_VEL
LIN {X 0,Y 215.906,Z 1177.641,A -85,B 0,C 180,E1 8778.609,E2 8778.609} C_VEL
LIN {X 0,Y 207.102,Z 1184.018,A -85,B 0,C 180,E1 8772.524,E2 8772.524} C_VEL
LIN {X 0,Y 200.677,Z 1188.937,A -85,B 0,C 180,E1 8766.364,E2 8766.364} C_VEL
LIN {X 0,Y 196.171,Z 1192.756,A -85,B 0,C 180,E1 8759.945,E2 8759.945} C_VEL
LIN {X 0,Y 193.38,Z 1195.593,A -85,B 0,C 180,E1 8753.138,E2 8753.138} C_VEL
LIN {X 0,Y 192.149,Z 1197.437,A -85,B 0,C 180,E1 8745.699,E2 8745.699} C_VEL
LIN {X 0,Y 191.929,Z 1197.905,A -85,B 0,C 180,E1 8739.294,E2 8739.294} C_VEL
LIN {X 0,Y 191.925,Z 1197.465,A -85,B 0,C 180,E1 8733.584,E2 8733.584} C_VEL
LIN {X 0,Y 192.184,Z 1196.056,A -85,B 0,C 180,E1 8727.316,E2 8727.316} C_VEL
LIN {X 0,Y 193.537,Z 1193.024,A -85,B 0,C 180,E1 8719.883,E2 8719.883} C_VEL
LIN {X 0,Y 196.247,Z 1189.247,A -85,B 0,C 180,E1 8713.422,E2 8713.422} C_VEL
LIN {X 0,Y 200.496,Z 1184.525,A -85,B 0,C 180,E1 8707.311,E2 8707.311} C_VEL
LIN {X 0,Y 206.51,Z 1178.636,A -85,B 0,C 180,E1 8701.359,E2 8701.359} C_VEL
LIN {X 0,Y 214.422,Z 1171.453,A -85,B 0,C 180,E1 8695.628,E2 8695.628} C_VEL
LIN {X 0,Y 226.348,Z 1160.996,A -85,B 0,C 180,E1 8689.174,E2 8689.174} C_VEL
LIN {X 0,Y 238.914,Z 1149.835,A -85,B 0,C 180,E1 8683.961,E2 8683.961} C_VEL
LIN {X 0,Y 250.615,Z 1139.251,A -85,B 0,C 180,E1 8680.004,E2 8680.004} C_VEL
LIN {X 0,Y 263.318,Z 1127.356,A -85,B 0,C 180,E1 8676.39,E2 8676.39} C_VEL
LIN {X 0,Y 279.705,Z 1111.199,A -85,B 0,C 180,E1 8672.475,E2 8672.475} C_VEL
LIN {X 0,Y 294.933,Z 1094.93,A -85,B 0,C 180,E1 8669.395,E2 8669.395} C_VEL
LIN {X 0,Y 307.81,Z 1080.281,A -85,B 0,C 180,E1 8667.123,E2 8667.123} C_VEL
LIN {X 0,Y 321.114,Z 1064.066,A -85,B 0,C 180,E1 8665.03,E2 8665.03} C_VEL
LIN {X 0,Y 336.429,Z 1043.837,A -85,B 0,C 180,E1 8662.882,E2 8662.882} C_VEL
LIN {X 0,Y 350.468,Z 1023.082,A -85,B 0,C 180,E1 8661.108,E2 8661.108} C_VEL
LIN {X 0,Y 361.715,Z 1004.879,A -85,B 0,C 180,E1 8659.804,E2 8659.804} C_VEL
LIN {X 0,Y 372.075,Z 986.506,A -85,B 0,C 180,E1 8658.693,E2 8658.693} C_VEL
LIN {X 0,Y 382.317,Z 966.411,A -85,B 0,C 180,E1 8657.661,E2 8657.661} C_VEL
LIN {X 0,Y 394.26,Z 939.639,A -85,B 0,C 180,E1 8656.541,E2 8656.541} C_VEL
LIN {X 0,Y 402.803,Z 917.241,A -85,B 0,C 180,E1 8655.782,E2 8655.782} C_VEL
LIN {X 0,Y 409.541,Z 896.884,A -85,B 0,C 180,E1 8655.211,E2 8655.211} C_VEL
LIN {X 0,Y 415.627,Z 875.32,A -85,B 0,C 180,E1 8654.71,E2 8654.71} C_VEL
LIN {X 0,Y 421.83,Z 848.418,A -85,B 0,C 180,E1 8654.218,E2 8654.218} C_VEL
LIN {X 0,Y 426.197,Z 821.485,A -85,B 0,C 180,E1 8653.813,E2 8653.813} C_VEL
LIN {X 0,Y 441.573,Z 681.786,A -85,B 0,C 180,E1 8651.911,E2 8651.911} C_VEL
LIN {X 0,Y 445.573,Z 645.065,A -85,B 0,C 180,E1 8651.39,E2 8651.39} C_VEL
LIN {X 0,Y 444.199,Z 641.901,A -85,B 0,C 180,E1 8649.458,E2 8649.458} C_VEL
LIN {X 0,Y 442.996,Z 638.709,A -85,B 0,C 180,E1 8646.871,E2 8646.871} C_VEL
LIN {X 0,Y 442.654,Z 638.352,A -85,B 0,C 180,E1 8645.83,E2 8645.83} C_VEL
LIN {X 0,Y 442.333,Z 639.082,A -85,B 0,C 180,E1 8644.831,E2 8644.831} C_VEL
LIN {X 0,Y 441.577,Z 645.671,A -85,B 0,C 180,E1 8641.975,E2 8641.975} C_VEL
LIN {X 0,Y 441.662,Z 646.287,A -85,B 0,C 180,E1 8641.327,E2 8641.327} C_VEL
LIN {X 0,Y 442.091,Z 646.911,A -85,B 0,C 180,E1 8640,E2 8640} C_VEL
LIN {X 0,Y 443.73,Z 651.173,A -85,B 0,C 180,E1 8636.835,E2 8636.835} C_VEL
